LIN {X 0,Y 166.434,Z 455.503,A -85,B 0,C 180,E1 -24153.296,E2 -24153.296} C_VEL
LIN {X 0,Y 169.593,Z 462.541,A -85,B 0,C 180,E1 -24157.756,E2 -24157.756} C_VEL
LIN {X 0,Y 171.925,Z 468.212,A -85,B 0,C 180,E1 -24160.849,E2 -24160.849} C_VEL
LIN {X 0,Y 174.056,Z 474.701,A -85,B 0,C 180,E1 -24163.902,E2 -24163.902} C_VEL
LIN {X 0,Y 175.584,Z 481.015,A -85,B 0,C 180,E1 -24166.592,E2 -24166.592} C_VEL
LIN {X 0,Y 174.825,Z 487.861,A -85,B 0,C 180,E1 -24168.642,E2 -24168.642} C_VEL
LIN {X 0,Y 172.622,Z 497.216,A -85,B 0,C 180,E1 -24171.532,E2 -24171.532} C_VEL
LIN {X 0,Y 170.129,Z 504.353,A -85,B 0,C 180,E1 -24173.945,E2 -24173.945} C_VEL
LIN {X 0,Y 165.916,Z 511.785,A -85,B 0,C 180,E1 -24176.595,E2 -24176.595} C_VEL
LIN {X 0,Y 161.161,Z 519.066,A -85,B 0,C 180,E1 -24179.908,E2 -24179.908} C_VEL
LIN {X 0,Y 157.26,Z 524.869,A -85,B 0,C 180,E1 -24183.462,E2 -24183.462} C_VEL
LIN {X 0,Y 153.991,Z 529.408,A -85,B 0,C 180,E1 -24187.181,E2 -24187.181} C_VEL
LIN {X 0,Y 151.34,Z 532.851,A -85,B 0,C 180,E1 -24191.037,E2 -24191.037} C_VEL
LIN {X 0,Y 149.93,Z 534.573,A -85,B 0,C 180,E1 -24193.672,E2 -24193.672} C_VEL
LIN {X 0,Y 148.978,Z 535.901,A -85,B 0,C 180,E1 -24196.363,E2 -24196.363} C_VEL
LIN {X 0,Y 148.309,Z 536.803,A -85,B 0,C 180,E1 -24199.08,E2 -24199.08} C_VEL
LIN {X 0,Y 147.919,Z 537.372,A -85,B 0,C 180,E1 -24204.553,E2 -24204.553} C_VEL
LIN {X 0,Y 147.968,Z 537.384,A -85,B 0,C 180,E1 -24205.296,E2 -24205.296} C_VEL
LIN {X 0,Y 148.105,Z 541.561,A -85,B 0,C 180,E1 -24210.006,E2 -24210.006} C_VEL
LIN {X 0,Y 147.802,Z 543.506,A -85,B 0,C 180,E1 -24213.069,E2 -24213.069} C_VEL
LIN {X 0,Y 147.952,Z 545.577,A -85,B 0,C 180,E1 -24218.199,E2 -24218.199} C_VEL
LIN {X 0,Y 149.306,Z 546.349,A -85,B 0,C 180,E1 -24223.618,E2 -24223.618} C_VEL
LIN {X 0,Y 151.84,Z 545.71,A -85,B 0,C 180,E1 -24228.911,E2 -24228.911} C_VEL
LIN {X 0,Y 155.965,Z 543.606,A -85,B 0,C 180,E1 -24233.931,E2 -24233.931} C_VEL
LIN {X 0,Y 161.202,Z 540.049,A -85,B 0,C 180,E1 -24238.663,E2 -24238.663} C_VEL
LIN {X 0,Y 165.955,Z 536.223,A -85,B 0,C 180,E1 -24242.114,E2 -24242.114} C_VEL
LIN {X 0,Y 171.027,Z 531.735,A -85,B 0,C 180,E1 -24245.126,E2 -24245.126} C_VEL
LIN {X 0,Y 177.232,Z 525.759,A -85,B 0,C 180,E1 -24248.092,E2 -24248.092} C_VEL
LIN {X 0,Y 179.758,Z 522.779,A -85,B 0,C 180,E1 -24249.524,E2 -24249.524} C_VEL
LIN {X 0,Y 182.55,Z 517.989,A -85,B 0,C 180,E1 -24252.134,E2 -24252.134} C_VEL
LIN {X 0,Y 185.7,Z 511.799,A -85,B 0,C 180,E1 -24255.202,E2 -24255.202} C_VEL
LIN {X 0,Y 187.148,Z 509.452,A -85,B 0,C 180,E1 -24256.096,E2 -24256.096} C_VEL
LIN {X 0,Y 188.812,Z 506.875,A -85,B 0,C 180,E1 -24257.01,E2 -24257.01} C_VEL
LIN {X 0,Y 189.502,Z 504.868,A -85,B 0,C 180,E1 -24258.12,E2 -24258.12} C_VEL
LIN {X 0,Y 189.981,Z 501.234,A -85,B 0,C 180,E1 -24261.031,E2 -24261.031} C_VEL
LIN {X 0,Y 189.707,Z 499.154,A -85,B 0,C 180,E1 -24263.647,E2 -24263.647} C_VEL
LIN {X 0,Y 189.489,Z 497.804,A -85,B 0,C 180,E1 -24266.196,E2 -24266.196} C_VEL
LIN {X 0,Y 189.328,Z 496.956,A -85,B 0,C 180,E1 -24268.688,E2 -24268.688} C_VEL
LIN {X 0,Y 189.184,Z 496.682,A -85,B 0,C 180,E1 -24271.122,E2 -24271.122} C_VEL
LIN {X 0,Y 188.92,Z 497.163,A -85,B 0,C 180,E1 -24273.485,E2 -24273.485} C_VEL
LIN {X 0,Y 188.706,Z 498.014,A -85,B 0,C 180,E1 -24275.815,E2 -24275.815} C_VEL
LIN {X 0,Y 188.644,Z 499.613,A -85,B 0,C 180,E1 -24278.661,E2 -24278.661} C_VEL
LIN {X 0,Y 188.327,Z 502.026,A -85,B 0,C 180,E1 -24281.505,E2 -24281.505} C_VEL
LIN {X 0,Y 187.812,Z 504.455,A -85,B 0,C 180,E1 -24283.7,E2 -24283.7} C_VEL
LIN {X 0,Y 187.108,Z 506.134,A -85,B 0,C 180,E1 -24284.755,E2 -24284.755} C_VEL
LIN {X 0,Y 183.978,Z 511.853,A -85,B 0,C 180,E1 -24287.871,E2 -24287.871} C_VEL
LIN {X 0,Y 183.305,Z 512.868,A -85,B 0,C 180,E1 -24288.387,E2 -24288.387} C_VEL
LIN {X 0,Y 175.523,Z 520.816,A -85,B 0,C 180,E1 -24291.364,E2 -24291.364} C_VEL
LIN {X 0,Y 169.603,Z 526.103,A -85,B 0,C 180,E1 -24294.032,E2 -24294.032} C_VEL
LIN {X 0,Y 162.956,Z 531.203,A -85,B 0,C 180,E1 -24297.527,E2 -24297.527} C_VEL
LIN {X 0,Y 157.198,Z 535.016,A -85,B 0,C 180,E1 -24301.28,E2 -24301.28} C_VEL
LIN {X 0,Y 152.28,Z 537.685,A -85,B 0,C 180,E1 -24305.295,E2 -24305.295} C_VEL
LIN {X 0,Y 149.19,Z 538.988,A -85,B 0,C 180,E1 -24308.374,E2 -24308.374} C_VEL
LIN {X 0,Y 146.941,Z 539.635,A -85,B 0,C 180,E1 -24311.029,E2 -24311.029} C_VEL
LIN {X 0,Y 144.854,Z 539.91,A -85,B 0,C 180,E1 -24314.038,E2 -24314.038} C_VEL
LIN {X 0,Y 143.177,Z 539.754,A -85,B 0,C 180,E1 -24317.128,E2 -24317.128} C_VEL
LIN {X 0,Y 141.877,Z 539.109,A -85,B 0,C 180,E1 -24320.288,E2 -24320.288} C_VEL
LIN {X 0,Y 140.475,Z 536.929,A -85,B 0,C 180,E1 -24325.759,E2 -24325.759} C_VEL
LIN {X 0,Y 140.134,Z 533.138,A -85,B 0,C 180,E1 -24331.496,E2 -24331.496} C_VEL
LIN {X 0,Y 140.646,Z 527.91,A -85,B 0,C 180,E1 -24336.908,E2 -24336.908} C_VEL
LIN {X 0,Y 141.633,Z 521.475,A -85,B 0,C 180,E1 -24341.891,E2 -24341.891} C_VEL
LIN {X 0,Y 143.083,Z 513.619,A -85,B 0,C 180,E1 -24346.548,E2 -24346.548} C_VEL
LIN {X 0,Y 144.81,Z 505.438,A -85,B 0,C 180,E1 -24350.393,E2 -24350.393} C_VEL
LIN {X 0,Y 146.926,Z 496.371,A -85,B 0,C 180,E1 -24353.82,E2 -24353.82} C_VEL
LIN {X 0,Y 149.55,Z 484.775,A -85,B 0,C 180,E1 -24357.284,E2 -24357.284} C_VEL
LIN {X 0,Y 150.844,Z 478.491,A -85,B 0,C 180,E1 -24358.834,E2 -24358.834} C_VEL
LIN {X 0,Y 149.746,Z 466.485,A -85,B 0,C 180,E1 -24361.622,E2 -24361.622} C_VEL
LIN {X 0,Y 148.306,Z 454.178,A -85,B 0,C 180,E1 -24363.996,E2 -24363.996} C_VEL
LIN {X 0,Y 146.033,Z 439.457,A -85,B 0,C 180,E1 -24366.272,E2 -24366.272} C_VEL
LIN {X 0,Y 144.595,Z 431.334,A -85,B 0,C 180,E1 -24367.355,E2 -24367.355} C_VEL
LIN {X 0,Y 144.497,Z 428.599,A -85,B 0,C 180,E1 -24370.089,E2 -24370.089} C_VEL
LIN {X 0,Y 143.779,Z 424.334,A -85,B 0,C 180,E1 -24374.762,E2 -24374.762} C_VEL
LIN {X 0,Y 144.189,Z 426.576,A -85,B 0,C 180,E1 -24378.751,E2 -24378.751} C_VEL
LIN {X 0,Y 144.55,Z 428.254,A -85,B 0,C 180,E1 -24381.607,E2 -24381.607} C_VEL
LIN {X 0,Y 145.11,Z 431.41,A -85,B 0,C 180,E1 -24386.349,E2 -24386.349} C_VEL
LIN {X 0,Y 147.226,Z 438.421,A -85,B 0,C 180,E1 -24387.563,E2 -24387.563} C_VEL
LIN {X 0,Y 149.67,Z 450.103,A -85,B 0,C 180,E1 -24389.729,E2 -24389.729} C_VEL
LIN {X 0,Y 151.023,Z 459.538,A -85,B 0,C 180,E1 -24391.761,E2 -24391.761} C_VEL
LIN {X 0,Y 151.915,Z 469.677,A -85,B 0,C 180,E1 -24394.305,E2 -24394.305} C_VEL
LIN {X 0,Y 152.07,Z 476.634,A -85,B 0,C 180,E1 -24396.296,E2 -24396.296} C_VEL
LIN {X 0,Y 149.516,Z 486.319,A -85,B 0,C 180,E1 -24399.217,E2 -24399.217} C_VEL
LIN {X 0,Y 147.124,Z 494.539,A -85,B 0,C 180,E1 -24402.407,E2 -24402.407} C_VEL
LIN {X 0,Y 145.091,Z 501.591,A -85,B 0,C 180,E1 -24405.871,E2 -24405.871} C_VEL
LIN {X 0,Y 143.101,Z 508.264,A -85,B 0,C 180,E1 -24410.1,E2 -24410.1} C_VEL
LIN {X 0,Y 141.677,Z 513.845,A -85,B 0,C 180,E1 -24414.873,E2 -24414.873} C_VEL
LIN {X 0,Y 140.813,Z 517.925,A -85,B 0,C 180,E1 -24419.932,E2 -24419.932} C_VEL
LIN {X 0,Y 140.738,Z 519.778,A -85,B 0,C 180,E1 -24423.311,E2 -24423.311} C_VEL
LIN {X 0,Y 141.111,Z 521.102,A -85,B 0,C 180,E1 -24427.169,E2 -24427.169} C_VEL
LIN {X 0,Y 142.415,Z 521.578,A -85,B 0,C 180,E1 -24432.25,E2 -24432.25} C_VEL
LIN {X 0,Y 144.53,Z 520.651,A -85,B 0,C 180,E1 -24437.097,E2 -24437.097} C_VEL
LIN {X 0,Y 147.428,Z 518.388,A -85,B 0,C 180,E1 -24441.706,E2 -24441.706} C_VEL
LIN {X 0,Y 151.032,Z 514.814,A -85,B 0,C 180,E1 -24446.056,E2 -24446.056} C_VEL
LIN {X 0,Y 155.463,Z 509.711,A -85,B 0,C 180,E1 -24450.181,E2 -24450.181} C_VEL
LIN {X 0,Y 159.597,Z 504.413,A -85,B 0,C 180,E1 -24453.282,E2 -24453.282} C_VEL
LIN {X 0,Y 164.694,Z 496.927,A -85,B 0,C 180,E1 -24456.542,E2 -24456.542} C_VEL
LIN {X 0,Y 166.412,Z 493.936,A -85,B 0,C 180,E1 -24457.661,E2 -24457.661} C_VEL
LIN {X 0,Y 167.735,Z 487.888,A -85,B 0,C 180,E1 -24460.416,E2 -24460.416} C_VEL
LIN {X 0,Y 168.468,Z 480.689,A -85,B 0,C 180,E1 -24463.612,E2 -24463.612} C_VEL
LIN {X 0,Y 168.234,Z 475.376,A -85,B 0,C 180,E1 -24466.102,E2 -24466.102} C_VEL
LIN {X 0,Y 167.124,Z 469.966,A -85,B 0,C 180,E1 -24469.093,E2 -24469.093} C_VEL
LIN {X 0,Y 165.277,Z 464.338,A -85,B 0,C 180,E1 -24472.672,E2 -24472.672} C_VEL
LIN {X 0,Y 163.325,Z 459.565,A -85,B 0,C 180,E1 -24476.343,E2 -24476.343} C_VEL
LIN {X 0,Y 160.83,Z 453.807,A -85,B 0,C 180,E1 -24481.879,E2 -24481.879} C_VEL
LIN {X 0,Y 157.948,Z 450.631,A -85,B 0,C 180,E1 -24490.253,E2 -24490.253} C_VEL
LIN {X 0,Y 157.668,Z 450.184,A -85,B 0,C 180,E1 -24492.879,E2 -24492.879} C_VEL
LIN {X 0,Y 157.604,Z 450.264,A -85,B 0,C 180,E1 -24495.52,E2 -24495.52} C_VEL
LIN {X 0,Y 157.752,Z 450.92,A -85,B 0,C 180,E1 -24498.172,E2 -24498.172} C_VEL
LIN {X 0,Y 158.774,Z 453.562,A -85,B 0,C 180,E1 -24503.478,E2 -24503.478} C_VEL
LIN {X 0,Y 160.478,Z 455.834,A -85,B 0,C 180,E1 -24507.378,E2 -24507.378} C_VEL
LIN {X 0,Y 163.34,Z 462.175,A -85,B 0,C 180,E1 -24513.073,E2 -24513.073} C_VEL
LIN {X 0,Y 165.352,Z 467.137,A -85,B 0,C 180,E1 -24516.517,E2 -24516.517} C_VEL
LIN {X 0,Y 167.729,Z 474.013,A -85,B 0,C 180,E1 -24520.504,E2 -24520.504} C_VEL
LIN {X 0,Y 169.286,Z 479.911,A -85,B 0,C 180,E1 -24523.449,E2 -24523.449} C_VEL
LIN {X 0,Y 170.103,Z 484.114,A -85,B 0,C 180,E1 -24525.391,E2 -24525.391} C_VEL
LIN {X 0,Y 169.683,Z 487.961,A -85,B 0,C 180,E1 -24526.705,E2 -24526.705} C_VEL
LIN {X 0,Y 167.552,Z 496.578,A -85,B 0,C 180,E1 -24529.499,E2 -24529.499} C_VEL
LIN {X 0,Y 164.427,Z 505,A -85,B 0,C 180,E1 -24532.485,E2 -24532.485} C_VEL
LIN {X 0,Y 160.933,Z 510.894,A -85,B 0,C 180,E1 -24534.653,E2 -24534.653} C_VEL
LIN {X 0,Y 155.821,Z 518.232,A -85,B 0,C 180,E1 -24538.005,E2 -24538.005} C_VEL
LIN {X 0,Y 150.892,Z 524.956,A -85,B 0,C 180,E1 -24542.248,E2 -24542.248} C_VEL
LIN {X 0,Y 147.452,Z 529.377,A -85,B 0,C 180,E1 -24546.108,E2 -24546.108} C_VEL
LIN {X 0,Y 144.62,Z 532.715,A -85,B 0,C 180,E1 -24550.12,E2 -24550.12} C_VEL
LIN {X 0,Y 143.092,Z 534.383,A -85,B 0,C 180,E1 -24552.868,E2 -24552.868} C_VEL
LIN {X 0,Y 142.042,Z 535.645,A -85,B 0,C 180,E1 -24555.684,E2 -24555.684} C_VEL
LIN {X 0,Y 140.9,Z 536.888,A -85,B 0,C 180,E1 -24561.401,E2 -24561.401} C_VEL
LIN {X 0,Y 140.926,Z 537.009,A -85,B 0,C 180,E1 -24565.683,E2 -24565.683} C_VEL
LIN {X 0,Y 141.044,Z 540.777,A -85,B 0,C 180,E1 -24570.006,E2 -24570.006} C_VEL
LIN {X 0,Y 140.746,Z 544.03,A -85,B 0,C 180,E1 -24575.738,E2 -24575.738} C_VEL
LIN {X 0,Y 141.489,Z 545.788,A -85,B 0,C 180,E1 -24581.466,E2 -24581.466} C_VEL
LIN {X 0,Y 143.556,Z 546.056,A -85,B 0,C 180,E1 -24587.088,E2 -24587.088} C_VEL
LIN {X 0,Y 147.13,Z 544.937,A -85,B 0,C 180,E1 -24592.472,E2 -24592.472} C_VEL
LIN {X 0,Y 152.123,Z 542.393,A -85,B 0,C 180,E1 -24597.522,E2 -24597.522} C_VEL
LIN {X 0,Y 158.161,Z 538.375,A -85,B 0,C 180,E1 -24602.23,E2 -24602.23} C_VEL
LIN {X 0,Y 165.332,Z 532.771,A -85,B 0,C 180,E1 -24606.527,E2 -24606.527} C_VEL
LIN {X 0,Y 173.738,Z 525.291,A -85,B 0,C 180,E1 -24610.339,E2 -24610.339} C_VEL
LIN {X 0,Y 181.682,Z 517.009,A -85,B 0,C 180,E1 -24613.369,E2 -24613.369} C_VEL
LIN {X 0,Y 187.148,Z 509.452,A -85,B 0,C 180,E1 -24616.096,E2 -24616.096} C_VEL
LIN {X 0,Y 188.189,Z 507.429,A -85,B 0,C 180,E1 -24617.029,E2 -24617.029} C_VEL
LIN {X 0,Y 188.45,Z 505.993,A -85,B 0,C 180,E1 -24618.115,E2 -24618.115} C_VEL
LIN {X 0,Y 187.888,Z 504.71,A -85,B 0,C 180,E1 -24619.879,E2 -24619.879} C_VEL
LIN {X 0,Y 185.048,Z 503.736,A -85,B 0,C 180,E1 -24624.404,E2 -24624.404} C_VEL
LIN {X 0,Y 184.695,Z 503.307,A -85,B 0,C 180,E1 -24625.736,E2 -24625.736} C_VEL
LIN {X 0,Y 184.575,Z 502.51,A -85,B 0,C 180,E1 -24627.786,E2 -24627.786} C_VEL
LIN {X 0,Y 184.432,Z 501.995,A -85,B 0,C 180,E1 -24631.224,E2 -24631.224} C_VEL
LIN {X 0,Y 183.919,Z 502.999,A -85,B 0,C 180,E1 -24635.143,E2 -24635.143} C_VEL
LIN {X 0,Y 183.755,Z 504.095,A -85,B 0,C 180,E1 -24637.513,E2 -24637.513} C_VEL
LIN {X 0,Y 183.185,Z 506.581,A -85,B 0,C 180,E1 -24640.966,E2 -24640.966} C_VEL
LIN {X 0,Y 182.92,Z 507.664,A -85,B 0,C 180,E1 -24642.098,E2 -24642.098} C_VEL
LIN {X 0,Y 182.361,Z 508.953,A -85,B 0,C 180,E1 -24643.199,E2 -24643.199} C_VEL
LIN {X 0,Y 180.23,Z 512.392,A -85,B 0,C 180,E1 -24645.317,E2 -24645.317} C_VEL
LIN {X 0,Y 178.364,Z 515.141,A -85,B 0,C 180,E1 -24646.904,E2 -24646.904} C_VEL
LIN {X 0,Y 170.622,Z 522.314,A -85,B 0,C 180,E1 -24649.744,E2 -24649.744} C_VEL
LIN {X 0,Y 162.801,Z 528.59,A -85,B 0,C 180,E1 -24653.201,E2 -24653.201} C_VEL
LIN {X 0,Y 157.134,Z 532.454,A -85,B 0,C 180,E1 -24656.152,E2 -24656.152} C_VEL
LIN {X 0,Y 151.083,Z 535.98,A -85,B 0,C 180,E1 -24659.999,E2 -24659.999} C_VEL
LIN {X 0,Y 147.516,Z 537.697,A -85,B 0,C 180,E1 -24662.73,E2 -24662.73} C_VEL
LIN {X 0,Y 141.971,Z 539.667,A -85,B 0,C 180,E1 -24668.049,E2 -24668.049} C_VEL
LIN {X 0,Y 137.613,Z 540.109,A -85,B 0,C 180,E1 -24673.968,E2 -24673.968} C_VEL
LIN {X 0,Y 134.76,Z 538.93,A -85,B 0,C 180,E1 -24680.144,E2 -24680.144} C_VEL
LIN {X 0,Y 133.305,Z 536.181,A -85,B 0,C 180,E1 -24686.317,E2 -24686.317} C_VEL
LIN {X 0,Y 133.078,Z 531.96,A -85,B 0,C 180,E1 -24692.32,E2 -24692.32} C_VEL
LIN {X 0,Y 133.53,Z 527.733,A -85,B 0,C 180,E1 -24696.685,E2 -24696.685} C_VEL
LIN {X 0,Y 134.514,Z 521.399,A -85,B 0,C 180,E1 -24701.77,E2 -24701.77} C_VEL
LIN {X 0,Y 135.85,Z 513.969,A -85,B 0,C 180,E1 -24706.407,E2 -24706.407} C_VEL
LIN {X 0,Y 137.667,Z 505.685,A -85,B 0,C 180,E1 -24710.536,E2 -24710.536} C_VEL
LIN {X 0,Y 139.814,Z 496.657,A -85,B 0,C 180,E1 -24714.148,E2 -24714.148} C_VEL
LIN {X 0,Y 142.439,Z 485.41,A -85,B 0,C 180,E1 -24717.704,E2 -24717.704} C_VEL
LIN {X 0,Y 143.815,Z 478.396,A -85,B 0,C 180,E1 -24719.529,E2 -24719.529} C_VEL
LIN {X 0,Y 142.755,Z 466.616,A -85,B 0,C 180,E1 -24722.393,E2 -24722.393} C_VEL
LIN {X 0,Y 141.42,Z 454.741,A -85,B 0,C 180,E1 -24724.79,E2 -24724.79} C_VEL
LIN {X 0,Y 139.283,Z 440.562,A -85,B 0,C 180,E1 -24727.099,E2 -24727.099} C_VEL
LIN {X 0,Y 137.609,Z 431.53,A -85,B 0,C 180,E1 -24728.365,E2 -24728.365} C_VEL
LIN {X 0,Y 137.213,Z 428.007,A -85,B 0,C 180,E1 -24732.096,E2 -24732.096} C_VEL
LIN {X 0,Y 136.825,Z 425.791,A -85,B 0,C 180,E1 -24734.636,E2 -24734.636} C_VEL
LIN {X 0,Y 137.532,Z 429.376,A -85,B 0,C 180,E1 -24741.175,E2 -24741.175} C_VEL
LIN {X 0,Y 137.868,Z 431.391,A -85,B 0,C 180,E1 -24744.601,E2 -24744.601} C_VEL
LIN {X 0,Y 139.322,Z 434.977,A -85,B 0,C 180,E1 -24745.367,E2 -24745.367} C_VEL
LIN {X 0,Y 141.065,Z 440.756,A -85,B 0,C 180,E1 -24746.493,E2 -24746.493} C_VEL
LIN {X 0,Y 143.374,Z 452.691,A -85,B 0,C 180,E1 -24748.939,E2 -24748.939} C_VEL
LIN {X 0,Y 144.738,Z 463.608,A -85,B 0,C 180,E1 -24751.536,E2 -24751.536} C_VEL
LIN {X 0,Y 145.317,Z 474.217,A -85,B 0,C 180,E1 -24754.501,E2 -24754.501} C_VEL
LIN {X 0,Y 145.23,Z 477.614,A -85,B 0,C 180,E1 -24755.548,E2 -24755.548} C_VEL
LIN {X 0,Y 142.664,Z 486.874,A -85,B 0,C 180,E1 -24758.492,E2 -24758.492} C_VEL
LIN {X 0,Y 139.841,Z 496.127,A -85,B 0,C 180,E1 -24762.326,E2 -24762.326} C_VEL
LIN {X 0,Y 137.573,Z 503.587,A -85,B 0,C 180,E1 -24766.37,E2 -24766.37} C_VEL
LIN {X 0,Y 135.584,Z 510.216,A -85,B 0,C 180,E1 -24771.091,E2 -24771.091} C_VEL
LIN {X 0,Y 134.33,Z 515.09,A -85,B 0,C 180,E1 -24775.843,E2 -24775.843} C_VEL
LIN {X 0,Y 133.733,Z 518.16,A -85,B 0,C 180,E1 -24779.942,E2 -24779.942} C_VEL
LIN {X 0,Y 133.765,Z 520.802,A -85,B 0,C 180,E1 -24785.297,E2 -24785.297} C_VEL
LIN {X 0,Y 134.319,Z 521.728,A -85,B 0,C 180,E1 -24788.884,E2 -24788.884} C_VEL
LIN {X 0,Y 135.717,Z 521.998,A -85,B 0,C 180,E1 -24793.534,E2 -24793.534} C_VEL
LIN {X 0,Y 138.117,Z 520.976,A -85,B 0,C 180,E1 -24798.587,E2 -24798.587} C_VEL
LIN {X 0,Y 141.308,Z 518.673,A -85,B 0,C 180,E1 -24803.359,E2 -24803.359} C_VEL
LIN {X 0,Y 145.265,Z 515.006,A -85,B 0,C 180,E1 -24807.848,E2 -24807.848} C_VEL
LIN {X 0,Y 150.096,Z 509.817,A -85,B 0,C 180,E1 -24812.081,E2 -24812.081} C_VEL
LIN {X 0,Y 154.673,Z 504.25,A -85,B 0,C 180,E1 -24815.317,E2 -24815.317} C_VEL
LIN {X 0,Y 160.53,Z 495.958,A -85,B 0,C 180,E1 -24818.888,E2 -24818.888} C_VEL
LIN {X 0,Y 162.059,Z 490.288,A -85,B 0,C 180,E1 -24821.677,E2 -24821.677} C_VEL
LIN {X 0,Y 163.059,Z 483.358,A -85,B 0,C 180,E1 -24825.014,E2 -24825.014} C_VEL
LIN {X 0,Y 163.037,Z 478.55,A -85,B 0,C 180,E1 -24827.554,E2 -24827.554} C_VEL
LIN {X 0,Y 161.843,Z 472.685,A -85,B 0,C 180,E1 -24831.259,E2 -24831.259} C_VEL
LIN {X 0,Y 160.949,Z 469.202,A -85,B 0,C 180,E1 -24833.734,E2 -24833.734} C_VEL
LIN {X 0,Y 159.399,Z 464.755,A -85,B 0,C 180,E1 -24837.474,E2 -24837.474} C_VEL
LIN {X 0,Y 157.642,Z 459.938,A -85,B 0,C 180,E1 -24842.556,E2 -24842.556} C_VEL
LIN {X 0,Y 155.384,Z 457.237,A -85,B 0,C 180,E1 -24850.424,E2 -24850.424} C_VEL
LIN {X 0,Y 155.171,Z 456.816,A -85,B 0,C 180,E1 -24853.09,E2 -24853.09} C_VEL
LIN {X 0,Y 155.13,Z 457.006,A -85,B 0,C 180,E1 -24855.774,E2 -24855.774} C_VEL
LIN {X 0,Y 155.254,Z 457.742,A -85,B 0,C 180,E1 -24858.475,E2 -24858.475} C_VEL
LIN {X 0,Y 157.398,Z 462.06,A -85,B 0,C 180,E1 -24866.76,E2 -24866.76} C_VEL
LIN {X 0,Y 159.766,Z 468.365,A -85,B 0,C 180,E1 -24872.696,E2 -24872.696} C_VEL
LIN {X 0,Y 161.646,Z 474.19,A -85,B 0,C 180,E1 -24876.832,E2 -24876.832} C_VEL
LIN {X 0,Y 163.267,Z 479.692,A -85,B 0,C 180,E1 -24880.219,E2 -24880.219} C_VEL
LIN {X 0,Y 164.418,Z 485.714,A -85,B 0,C 180,E1 -24883.402,E2 -24883.402} C_VEL
LIN {X 0,Y 164.603,Z 488.774,A -85,B 0,C 180,E1 -24884.829,E2 -24884.829} C_VEL
LIN {X 0,Y 162.395,Z 496.794,A -85,B 0,C 180,E1 -24887.609,E2 -24887.609} C_VEL
LIN {X 0,Y 159.563,Z 504.092,A -85,B 0,C 180,E1 -24890.317,E2 -24890.317} C_VEL
LIN {X 0,Y 157.151,Z 508.602,A -85,B 0,C 180,E1 -24892.062,E2 -24892.062} C_VEL
LIN {X 0,Y 151.57,Z 516.352,A -85,B 0,C 180,E1 -24895.397,E2 -24895.397} C_VEL
LIN {X 0,Y 147.483,Z 521.585,A -85,B 0,C 180,E1 -24898.395,E2 -24898.395} C_VEL
LIN {X 0,Y 143.713,Z 526.242,A -85,B 0,C 180,E1 -24901.897,E2 -24901.897} C_VEL
LIN {X 0,Y 139.861,Z 530.55,A -85,B 0,C 180,E1 -24906.304,E2 -24906.304} C_VEL
LIN {X 0,Y 137.945,Z 532.58,A -85,B 0,C 180,E1 -24909.114,E2 -24909.114} C_VEL
LIN {X 0,Y 136.292,Z 534.197,A -85,B 0,C 180,E1 -24911.985,E2 -24911.985} C_VEL
LIN {X 0,Y 134.322,Z 536.12,A -85,B 0,C 180,E1 -24917.927,E2 -24917.927} C_VEL
LIN {X 0,Y 133.854,Z 536.499,A -85,B 0,C 180,E1 -24920.944,E2 -24920.944} C_VEL
LIN {X 0,Y 133.889,Z 536.308,A -85,B 0,C 180,E1 -24925.832,E2 -24925.832} C_VEL
LIN {X 0,Y 133.983,Z 539.877,A -85,B 0,C 180,E1 -24930.007,E2 -24930.007} C_VEL
LIN {X 0,Y 133.72,Z 541.858,A -85,B 0,C 180,E1 -24933.019,E2 -24933.019} C_VEL
LIN {X 0,Y 133.943,Z 544.554,A -85,B 0,C 180,E1 -24939.063,E2 -24939.063} C_VEL
LIN {X 0,Y 135.483,Z 545.791,A -85,B 0,C 180,E1 -24945.039,E2 -24945.039} C_VEL
LIN {X 0,Y 138.468,Z 545.628,A -85,B 0,C 180,E1 -24950.818,E2 -24950.818} C_VEL
LIN {X 0,Y 143.089,Z 544.04,A -85,B 0,C 180,E1 -24956.241,E2 -24956.241} C_VEL
LIN {X 0,Y 148.929,Z 541.073,A -85,B 0,C 180,E1 -24961.278,E2 -24961.278} C_VEL
LIN {X 0,Y 153.776,Z 537.996,A -85,B 0,C 180,E1 -24964.648,E2 -24964.648} C_VEL
LIN {X 0,Y 159.739,Z 533.768,A -85,B 0,C 180,E1 -24968.027,E2 -24968.027} C_VEL
LIN {X 0,Y 166.248,Z 528.644,A -85,B 0,C 180,E1 -24970.945,E2 -24970.945} C_VEL
LIN {X 0,Y 174.4,Z 521.267,A -85,B 0,C 180,E1 -24974.044,E2 -24974.044} C_VEL
LIN {X 0,Y 177.84,Z 517.687,A -85,B 0,C 180,E1 -24975.349,E2 -24975.349} C_VEL
LIN {X 0,Y 183.011,Z 511.124,A -85,B 0,C 180,E1 -24977.838,E2 -24977.838} C_VEL
LIN {X 0,Y 184.001,Z 509.611,A -85,B 0,C 180,E1 -24978.482,E2 -24978.482} C_VEL
LIN {X 0,Y 184.504,Z 507.996,A -85,B 0,C 180,E1 -24979.642,E2 -24979.642} C_VEL
LIN {X 0,Y 184.815,Z 506.578,A -85,B 0,C 180,E1 -24980.933,E2 -24980.933} C_VEL
LIN {X 0,Y 184.926,Z 504.798,A -85,B 0,C 180,E1 -24982.955,E2 -24982.955} C_VEL
LIN {X 0,Y 184.695,Z 503.307,A -85,B 0,C 180,E1 -24985.736,E2 -24985.736} C_VEL
LIN {X 0,Y 184.093,Z 503.142,A -85,B 0,C 180,E1 -24987.559,E2 -24987.559} C_VEL
LIN {X 0,Y 182.876,Z 503.911,A -85,B 0,C 180,E1 -24989.363,E2 -24989.363} C_VEL
LIN {X 0,Y 179.151,Z 507.539,A -85,B 0,C 180,E1 -24994.22,E2 -24994.22} C_VEL
LIN {X 0,Y 178.754,Z 508.182,A -85,B 0,C 180,E1 -24995.496,E2 -24995.496} C_VEL
LIN {X 0,Y 178.617,Z 508.687,A -85,B 0,C 180,E1 -24996.829,E2 -24996.829} C_VEL
LIN {X 0,Y 178.191,Z 510.04,A -85,B 0,C 180,E1 -24999.208,E2 -24999.208} C_VEL
LIN {X 0,Y 177.492,Z 511.907,A -85,B 0,C 180,E1 -25001.531,E2 -25001.531} C_VEL
LIN {X 0,Y 176.68,Z 513.237,A -85,B 0,C 180,E1 -25002.641,E2 -25002.641} C_VEL
LIN {X 0,Y 173.493,Z 517.348,A -85,B 0,C 180,E1 -25005.333,E2 -25005.333} C_VEL
LIN {X 0,Y 165.05,Z 524.498,A -85,B 0,C 180,E1 -25008.36,E2 -25008.36} C_VEL
LIN {X 0,Y 156.048,Z 530.857,A -85,B 0,C 180,E1 -25012.264,E2 -25012.264} C_VEL
LIN {X 0,Y 151.393,Z 533.632,A -85,B 0,C 180,E1 -25014.672,E2 -25014.672} C_VEL
LIN {X 0,Y 147.114,Z 535.919,A -85,B 0,C 180,E1 -25017.261,E2 -25017.261} C_VEL
LIN {X 0,Y 140.654,Z 538.692,A -85,B 0,C 180,E1 -25021.955,E2 -25021.955} C_VEL
LIN {X 0,Y 134.757,Z 540.203,A -85,B 0,C 180,E1 -25027.692,E2 -25027.692} C_VEL
LIN {X 0,Y 130.339,Z 540.171,A -85,B 0,C 180,E1 -25033.91,E2 -25033.91} C_VEL
LIN {X 0,Y 127.509,Z 538.489,A -85,B 0,C 180,E1 -25040.43,E2 -25040.43} C_VEL
LIN {X 0,Y 126.131,Z 535.301,A -85,B 0,C 180,E1 -25046.923,E2 -25046.923} C_VEL
LIN {X 0,Y 125.977,Z 531.907,A -85,B 0,C 180,E1 -25051.691,E2 -25051.691} C_VEL
LIN {X 0,Y 126.578,Z 526.199,A -85,B 0,C 180,E1 -25057.643,E2 -25057.643} C_VEL
LIN {X 0,Y 127.718,Z 519.453,A -85,B 0,C 180,E1 -25062.975,E2 -25062.975} C_VEL
LIN {X 0,Y 129.053,Z 512.468,A -85,B 0,C 180,E1 -25067.321,E2 -25067.321} C_VEL
LIN {X 0,Y 131.034,Z 503.675,A -85,B 0,C 180,E1 -25071.688,E2 -25071.688} C_VEL
LIN {X 0,Y 133.377,Z 494.169,A -85,B 0,C 180,E1 -25075.462,E2 -25075.462} C_VEL
LIN {X 0,Y 136.004,Z 483.3,A -85,B 0,C 180,E1 -25078.879,E2 -25078.879} C_VEL
LIN {X 0,Y 136.784,Z 478.378,A -85,B 0,C 180,E1 -25080.206,E2 -25080.206} C_VEL
LIN {X 0,Y 135.756,Z 466.195,A -85,B 0,C 180,E1 -25083.302,E2 -25083.302} C_VEL
LIN {X 0,Y 134.388,Z 453.971,A -85,B 0,C 180,E1 -25085.874,E2 -25085.874} C_VEL
LIN {X 0,Y 132.271,Z 440.078,A -85,B 0,C 180,E1 -25088.261,E2 -25088.261} C_VEL
LIN {X 0,Y 130.572,Z 431.669,A -85,B 0,C 180,E1 -25089.514,E2 -25089.514} C_VEL
LIN {X 0,Y 129.898,Z 427.259,A -85,B 0,C 180,E1 -25094.48,E2 -25094.48} C_VEL
LIN {X 0,Y 130.516,Z 430.506,A -85,B 0,C 180,E1 -25100.697,E2 -25100.697} C_VEL
LIN {X 0,Y 130.674,Z 431.638,A -85,B 0,C 180,E1 -25102.752,E2 -25102.752} C_VEL
LIN {X 0,Y 132.142,Z 435.222,A -85,B 0,C 180,E1 -25103.595,E2 -25103.595} C_VEL
LIN {X 0,Y 134.561,Z 441.41,A -85,B 0,C 180,E1 -25105.032,E2 -25105.032} C_VEL
LIN {X 0,Y 136.861,Z 453.788,A -85,B 0,C 180,E1 -25107.73,E2 -25107.73} C_VEL
LIN {X 0,Y 137.937,Z 462.783,A -85,B 0,C 180,E1 -25109.994,E2 -25109.994} C_VEL
LIN {X 0,Y 138.556,Z 472.831,A -85,B 0,C 180,E1 -25112.901,E2 -25112.901} C_VEL
LIN {X 0,Y 138.425,Z 478.513,A -85,B 0,C 180,E1 -25114.726,E2 -25114.726} C_VEL
LIN {X 0,Y 135.54,Z 488.224,A -85,B 0,C 180,E1 -25118.023,E2 -25118.023} C_VEL
LIN {X 0,Y 133.075,Z 496.005,A -85,B 0,C 180,E1 -25121.416,E2 -25121.416} C_VEL
LIN {X 0,Y 130.713,Z 503.484,A -85,B 0,C 180,E1 -25125.587,E2 -25125.587} C_VEL
LIN {X 0,Y 128.729,Z 509.804,A -85,B 0,C 180,E1 -25130.214,E2 -25130.214} C_VEL
LIN {X 0,Y 127.526,Z 514.191,A -85,B 0,C 180,E1 -25134.406,E2 -25134.406} C_VEL
LIN {X 0,Y 126.648,Z 518.393,A -85,B 0,C 180,E1 -25139.953,E2 -25139.953} C_VEL
LIN {X 0,Y 126.554,Z 520.376,A -85,B 0,C 180,E1 -25143.724,E2 -25143.724} C_VEL
LIN {X 0,Y 127.319,Z 522.086,A -85,B 0,C 180,E1 -25149.396,E2 -25149.396} C_VEL
LIN {X 0,Y 129.123,Z 522.396,A -85,B 0,C 180,E1 -25155.027,E2 -25155.027} C_VEL
LIN {X 0,Y 131.812,Z 521.31,A -85,B 0,C 180,E1 -25160.223,E2 -25160.223} C_VEL
LIN {X 0,Y 135.887,Z 518.496,A -85,B 0,C 180,E1 -25165.83,E2 -25165.83} C_VEL
LIN {X 0,Y 139.682,Z 515.195,A -85,B 0,C 180,E1 -25169.793,E2 -25169.793} C_VEL
LIN {X 0,Y 144.967,Z 509.92,A -85,B 0,C 180,E1 -25174.132,E2 -25174.132} C_VEL
LIN {X 0,Y 149.983,Z 504.121,A -85,B 0,C 180,E1 -25177.49,E2 -25177.49} C_VEL
LIN {X 0,Y 154.677,Z 497.943,A -85,B 0,C 180,E1 -25180.209,E2 -25180.209} C_VEL
LIN {X 0,Y 156.141,Z 493.743,A -85,B 0,C 180,E1 -25182.436,E2 -25182.436} C_VEL
LIN {X 0,Y 157.574,Z 487.345,A -85,B 0,C 180,E1 -25185.801,E2 -25185.801} C_VEL
LIN {X 0,Y 157.888,Z 482.991,A -85,B 0,C 180,E1 -25188.281,E2 -25188.281} C_VEL
LIN {X 0,Y 157.117,Z 477.195,A -85,B 0,C 180,E1 -25192.289,E2 -25192.289} C_VEL
LIN {X 0,Y 156.027,Z 472.537,A -85,B 0,C 180,E1 -25196.127,E2 -25196.127} C_VEL
LIN {X 0,Y 154.895,Z 468.749,A -85,B 0,C 180,E1 -25200.001,E2 -25200.001} C_VEL
LIN {X 0,Y 154.3,Z 466.442,A -85,B 0,C 180,E1 -25202.611,E2 -25202.611} C_VEL
LIN {X 0,Y 152.464,Z 463.674,A -85,B 0,C 180,E1 -25210.626,E2 -25210.626} C_VEL
LIN {X 0,Y 152.243,Z 463.371,A -85,B 0,C 180,E1 -25214.235,E2 -25214.235} C_VEL
LIN {X 0,Y 152.269,Z 463.598,A -85,B 0,C 180,E1 -25216.078,E2 -25216.078} C_VEL
LIN {X 0,Y 152.364,Z 464.452,A -85,B 0,C 180,E1 -25218.838,E2 -25218.838} C_VEL
LIN {X 0,Y 153.324,Z 467.173,A -85,B 0,C 180,E1 -25224.365,E2 -25224.365} C_VEL
LIN {X 0,Y 154.196,Z 468.985,A -85,B 0,C 180,E1 -25227.116,E2 -25227.116} C_VEL
LIN {X 0,Y 155.54,Z 473.07,A -85,B 0,C 180,E1 -25231.306,E2 -25231.306} C_VEL
LIN {X 0,Y 157.302,Z 479.828,A -85,B 0,C 180,E1 -25236.478,E2 -25236.478} C_VEL
LIN {X 0,Y 158.571,Z 485.64,A -85,B 0,C 180,E1 -25240.221,E2 -25240.221} C_VEL
LIN {X 0,Y 159.132,Z 491.021,A -85,B 0,C 180,E1 -25243.252,E2 -25243.252} C_VEL
LIN {X 0,Y 158.588,Z 493.607,A -85,B 0,C 180,E1 -25244.297,E2 -25244.297} C_VEL
LIN {X 0,Y 155.575,Z 501.704,A -85,B 0,C 180,E1 -25247.351,E2 -25247.351} C_VEL
LIN {X 0,Y 152.552,Z 507.763,A -85,B 0,C 180,E1 -25249.845,E2 -25249.845} C_VEL
LIN {X 0,Y 146.731,Z 515.568,A -85,B 0,C 180,E1 -25253.231,E2 -25253.231} C_VEL
LIN {X 0,Y 141.493,Z 521.784,A -85,B 0,C 180,E1 -25256.89,E2 -25256.89} C_VEL
LIN {X 0,Y 137.168,Z 526.639,A -85,B 0,C 180,E1 -25260.803,E2 -25260.803} C_VEL
LIN {X 0,Y 133.363,Z 530.5,A -85,B 0,C 180,E1 -25265.073,E2 -25265.073} C_VEL
LIN {X 0,Y 131.32,Z 532.467,A -85,B 0,C 180,E1 -25268.007,E2 -25268.007} C_VEL
LIN {X 0,Y 129.535,Z 533.982,A -85,B 0,C 180,E1 -25271.01,E2 -25271.01} C_VEL
LIN {X 0,Y 127.354,Z 535.782,A -85,B 0,C 180,E1 -25277.255,E2 -25277.255} C_VEL
LIN {X 0,Y 126.83,Z 536.09,A -85,B 0,C 180,E1 -25280.438,E2 -25280.438} C_VEL
LIN {X 0,Y 126.842,Z 535.653,A -85,B 0,C 180,E1 -25286.116,E2 -25286.116} C_VEL
LIN {X 0,Y 126.924,Z 538.941,A -85,B 0,C 180,E1 -25290.007,E2 -25290.007} C_VEL
LIN {X 0,Y 126.68,Z 541.03,A -85,B 0,C 180,E1 -25293.187,E2 -25293.187} C_VEL
LIN {X 0,Y 126.937,Z 543.981,A -85,B 0,C 180,E1 -25299.568,E2 -25299.568} C_VEL
LIN {X 0,Y 128.619,Z 545.434,A -85,B 0,C 180,E1 -25305.862,E2 -25305.862} C_VEL
LIN {X 0,Y 131.855,Z 545.514,A -85,B 0,C 180,E1 -25311.914,E2 -25311.914} C_VEL
LIN {X 0,Y 136.744,Z 544.234,A -85,B 0,C 180,E1 -25317.559,E2 -25317.559} C_VEL
LIN {X 0,Y 142.926,Z 541.513,A -85,B 0,C 180,E1 -25322.751,E2 -25322.751} C_VEL
LIN {X 0,Y 150.227,Z 537.396,A -85,B 0,C 180,E1 -25327.464,E2 -25327.464} C_VEL
LIN {X 0,Y 156.485,Z 533.231,A -85,B 0,C 180,E1 -25330.64,E2 -25330.64} C_VEL
LIN {X 0,Y 163.372,Z 528.096,A -85,B 0,C 180,E1 -25333.501,E2 -25333.501} C_VEL
LIN {X 0,Y 171.956,Z 520.721,A -85,B 0,C 180,E1 -25336.513,E2 -25336.513} C_VEL
LIN {X 0,Y 178.389,Z 513.593,A -85,B 0,C 180,E1 -25339.363,E2 -25339.363} C_VEL
LIN {X 0,Y 179.01,Z 512.522,A -85,B 0,C 180,E1 -25340.034,E2 -25340.034} C_VEL
LIN {X 0,Y 179.52,Z 510.932,A -85,B 0,C 180,E1 -25341.54,E2 -25341.54} C_VEL
LIN {X 0,Y 179.677,Z 509.137,A -85,B 0,C 180,E1 -25344.075,E2 -25344.075} C_VEL
LIN {X 0,Y 179.594,Z 507.887,A -85,B 0,C 180,E1 -25346.779,E2 -25346.779} C_VEL
LIN {X 0,Y 179.476,Z 507.248,A -85,B 0,C 180,E1 -25349.491,E2 -25349.491} C_VEL
LIN {X 0,Y 179.29,Z 507.163,A -85,B 0,C 180,E1 -25351.94,E2 -25351.94} C_VEL
LIN {X 0,Y 178.754,Z 508.182,A -85,B 0,C 180,E1 -25355.496,E2 -25355.496} C_VEL
LIN {X 0,Y 178.11,Z 509.124,A -85,B 0,C 180,E1 -25356.704,E2 -25356.704} C_VEL
LIN {X 0,Y 176.799,Z 510.684,A -85,B 0,C 180,E1 -25357.811,E2 -25357.811} C_VEL
LIN {X 0,Y 172.261,Z 515.527,A -85,B 0,C 180,E1 -25360.65,E2 -25360.65} C_VEL
LIN {X 0,Y 171.363,Z 516.563,A -85,B 0,C 180,E1 -25361.435,E2 -25361.435} C_VEL
LIN {X 0,Y 169.464,Z 518.803,A -85,B 0,C 180,E1 -25363.123,E2 -25363.123} C_VEL
LIN {X 0,Y 168.323,Z 519.924,A -85,B 0,C 180,E1 -25363.82,E2 -25363.82} C_VEL
LIN {X 0,Y 161.461,Z 525.208,A -85,B 0,C 180,E1 -25366.148,E2 -25366.148} C_VEL
LIN {X 0,Y 153.267,Z 530.661,A -85,B 0,C 180,E1 -25369.43,E2 -25369.43} C_VEL
LIN {X 0,Y 145.759,Z 534.813,A -85,B 0,C 180,E1 -25373.076,E2 -25373.076} C_VEL
LIN {X 0,Y 139.135,Z 537.753,A -85,B 0,C 180,E1 -25377.104,E2 -25377.104} C_VEL
LIN {X 0,Y 133.578,Z 539.59,A -85,B 0,C 180,E1 -25381.283,E2 -25381.283} C_VEL
LIN {X 0,Y 127.549,Z 540.6,A -85,B 0,C 180,E1 -25387.297,E2 -25387.297} C_VEL
LIN {X 0,Y 123.069,Z 540.047,A -85,B 0,C 180,E1 -25393.854,E2 -25393.854} C_VEL
LIN {X 0,Y 120.309,Z 537.989,A -85,B 0,C 180,E1 -25400.517,E2 -25400.517} C_VEL
LIN {X 0,Y 118.991,Z 534.238,A -85,B 0,C 180,E1 -25407.618,E2 -25407.618} C_VEL
LIN {X 0,Y 118.922,Z 530.884,A -85,B 0,C 180,E1 -25412.131,E2 -25412.131} C_VEL
LIN {X 0,Y 119.57,Z 525.176,A -85,B 0,C 180,E1 -25418.108,E2 -25418.108} C_VEL
LIN {X 0,Y 120.667,Z 518.886,A -85,B 0,C 180,E1 -25423.182,E2 -25423.182} C_VEL
LIN {X 0,Y 122.284,Z 510.771,A -85,B 0,C 180,E1 -25428.342,E2 -25428.342} C_VEL
LIN {X 0,Y 124.438,Z 501.704,A -85,B 0,C 180,E1 -25432.914,E2 -25432.914} C_VEL
LIN {X 0,Y 126.958,Z 491.714,A -85,B 0,C 180,E1 -25436.851,E2 -25436.851} C_VEL
LIN {X 0,Y 129.805,Z 479.904,A -85,B 0,C 180,E1 -25440.505,E2 -25440.505} C_VEL
LIN {X 0,Y 128.957,Z 468.205,A -85,B 0,C 180,E1 -25443.71,E2 -25443.71} C_VEL
LIN {X 0,Y 127.756,Z 456.1,A -85,B 0,C 180,E1 -25446.488,E2 -25446.488} C_VEL
LIN {X 0,Y 125.9,Z 443.054,A -85,B 0,C 180,E1 -25448.932,E2 -25448.932} C_VEL
LIN {X 0,Y 124.303,Z 434.7,A -85,B 0,C 180,E1 -25450.27,E2 -25450.27} C_VEL
LIN {X 0,Y 123.429,Z 431.824,A -85,B 0,C 180,E1 -25450.774,E2 -25450.774} C_VEL
LIN {X 0,Y 122.982,Z 428.791,A -85,B 0,C 180,E1 -25454.449,E2 -25454.449} C_VEL
LIN {X 0,Y 123.581,Z 432.011,A -85,B 0,C 180,E1 -25460.738,E2 -25460.738} C_VEL
LIN {X 0,Y 124.959,Z 435.43,A -85,B 0,C 180,E1 -25461.584,E2 -25461.584} C_VEL
LIN {X 0,Y 128.493,Z 443.884,A -85,B 0,C 180,E1 -25463.85,E2 -25463.85} C_VEL
LIN {X 0,Y 130.448,Z 455.463,A -85,B 0,C 180,E1 -25466.59,E2 -25466.59} C_VEL
LIN {X 0,Y 131.418,Z 464.305,A -85,B 0,C 180,E1 -25468.985,E2 -25468.985} C_VEL
LIN {X 0,Y 131.899,Z 473.75,A -85,B 0,C 180,E1 -25471.902,E2 -25471.902} C_VEL
LIN {X 0,Y 131.658,Z 479.408,A -85,B 0,C 180,E1 -25473.819,E2 -25473.819} C_VEL
LIN {X 0,Y 128.958,Z 488.078,A -85,B 0,C 180,E1 -25476.893,E2 -25476.893} C_VEL
LIN {X 0,Y 126.368,Z 495.86,A -85,B 0,C 180,E1 -25480.406,E2 -25480.406} C_VEL
LIN {X 0,Y 124.253,Z 502.229,A -85,B 0,C 180,E1 -25484.017,E2 -25484.017} C_VEL
LIN {X 0,Y 122.166,Z 508.413,A -85,B 0,C 180,E1 -25488.437,E2 -25488.437} C_VEL
LIN {X 0,Y 120.46,Z 514.296,A -85,B 0,C 180,E1 -25494.096,E2 -25494.096} C_VEL
LIN {X 0,Y 119.539,Z 518.618,A -85,B 0,C 180,E1 -25499.996,E2 -25499.996} C_VEL
LIN {X 0,Y 119.621,Z 521.396,A -85,B 0,C 180,E1 -25505.971,E2 -25505.971} C_VEL
LIN {X 0,Y 120.488,Z 522.574,A -85,B 0,C 180,E1 -25510.689,E2 -25510.689} C_VEL
LIN {X 0,Y 122.569,Z 522.796,A -85,B 0,C 180,E1 -25516.524,E2 -25516.524} C_VEL
LIN {X 0,Y 125.609,Z 521.653,A -85,B 0,C 180,E1 -25522.016,E2 -25522.016} C_VEL
LIN {X 0,Y 129.49,Z 519.246,A -85,B 0,C 180,E1 -25527.13,E2 -25527.13} C_VEL
LIN {X 0,Y 134.315,Z 515.405,A -85,B 0,C 180,E1 -25531.907,E2 -25531.907} C_VEL
LIN {X 0,Y 140.04,Z 510.027,A -85,B 0,C 180,E1 -25536.33,E2 -25536.33} C_VEL
LIN {X 0,Y 145.012,Z 504.617,A -85,B 0,C 180,E1 -25539.482,E2 -25539.482} C_VEL
LIN {X 0,Y 149.309,Z 499.198,A -85,B 0,C 180,E1 -25542.001,E2 -25542.001} C_VEL
LIN {X 0,Y 151.314,Z 493.691,A -85,B 0,C 180,E1 -25545.202,E2 -25545.202} C_VEL
LIN {X 0,Y 152.395,Z 489.119,A -85,B 0,C 180,E1 -25547.852,E2 -25547.852} C_VEL
LIN {X 0,Y 152.601,Z 486.768,A -85,B 0,C 180,E1 -25549.385,E2 -25549.385} C_VEL
LIN {X 0,Y 152.256,Z 481.584,A -85,B 0,C 180,E1 -25553.374,E2 -25553.374} C_VEL
LIN {X 0,Y 151.529,Z 477.279,A -85,B 0,C 180,E1 -25557.343,E2 -25557.343} C_VEL
LIN {X 0,Y 150.599,Z 472.699,A -85,B 0,C 180,E1 -25562.676,E2 -25562.676} C_VEL
LIN {X 0,Y 149.916,Z 471.492,A -85,B 0,C 180,E1 -25565.381,E2 -25565.381} C_VEL
LIN {X 0,Y 149.133,Z 469.93,A -85,B 0,C 180,E1 -25570.866,E2 -25570.866} C_VEL
LIN {X 0,Y 149.034,Z 469.641,A -85,B 0,C 180,E1 -25573.639,E2 -25573.639} C_VEL
LIN {X 0,Y 149.005,Z 470.056,A -85,B 0,C 180,E1 -25576.44,E2 -25576.44} C_VEL
LIN {X 0,Y 149.38,Z 472.272,A -85,B 0,C 180,E1 -25582.111,E2 -25582.111} C_VEL
LIN {X 0,Y 149.964,Z 473.797,A -85,B 0,C 180,E1 -25584.948,E2 -25584.948} C_VEL
LIN {X 0,Y 150.935,Z 477.352,A -85,B 0,C 180,E1 -25589.27,E2 -25589.27} C_VEL
LIN {X 0,Y 151.532,Z 479.613,A -85,B 0,C 180,E1 -25591.547,E2 -25591.547} C_VEL
LIN {X 0,Y 152.656,Z 484.991,A -85,B 0,C 180,E1 -25595.944,E2 -25595.944} C_VEL
LIN {X 0,Y 153.443,Z 490.683,A -85,B 0,C 180,E1 -25599.885,E2 -25599.885} C_VEL
LIN {X 0,Y 153.625,Z 494.117,A -85,B 0,C 180,E1 -25601.988,E2 -25601.988} C_VEL
LIN {X 0,Y 152.709,Z 497.182,A -85,B 0,C 180,E1 -25603.334,E2 -25603.334} C_VEL
LIN {X 0,Y 149.614,Z 504.051,A -85,B 0,C 180,E1 -25606.152,E2 -25606.152} C_VEL
LIN {X 0,Y 146.245,Z 509.783,A -85,B 0,C 180,E1 -25608.65,E2 -25608.65} C_VEL
LIN {X 0,Y 140.136,Z 517.083,A -85,B 0,C 180,E1 -25612.104,E2 -25612.104} C_VEL
LIN {X 0,Y 135.586,Z 522.016,A -85,B 0,C 180,E1 -25615.246,E2 -25615.246} C_VEL
LIN {X 0,Y 131.411,Z 526.277,A -85,B 0,C 180,E1 -25618.839,E2 -25618.839} C_VEL
LIN {X 0,Y 126.94,Z 530.452,A -85,B 0,C 180,E1 -25623.718,E2 -25623.718} C_VEL
LIN {X 0,Y 124.745,Z 532.341,A -85,B 0,C 180,E1 -25626.782,E2 -25626.782} C_VEL
LIN {X 0,Y 121.383,Z 534.797,A -85,B 0,C 180,E1 -25633.18,E2 -25633.18} C_VEL
LIN {X 0,Y 120.414,Z 535.442,A -85,B 0,C 180,E1 -25636.507,E2 -25636.507} C_VEL
LIN {X 0,Y 119.614,Z 535.472,A -85,B 0,C 180,E1 -25643.259,E2 -25643.259} C_VEL
LIN {X 0,Y 119.817,Z 535.003,A -85,B 0,C 180,E1 -25646.455,E2 -25646.455} C_VEL
LIN {X 0,Y 119.872,Z 537.944,A -85,B 0,C 180,E1 -25650.007,E2 -25650.007} C_VEL
LIN {X 0,Y 119.642,Z 540.145,A -85,B 0,C 180,E1 -25653.375,E2 -25653.375} C_VEL
LIN {X 0,Y 119.954,Z 543.316,A -85,B 0,C 180,E1 -25660.131,E2 -25660.131} C_VEL
LIN {X 0,Y 121.791,Z 545.048,A -85,B 0,C 180,E1 -25666.777,E2 -25666.777} C_VEL
LIN {X 0,Y 125.299,Z 545.373,A -85,B 0,C 180,E1 -25673.125,E2 -25673.125} C_VEL
LIN {X 0,Y 130.477,Z 544.334,A -85,B 0,C 180,E1 -25679.005,E2 -25679.005} C_VEL
LIN {X 0,Y 137.027,Z 541.96,A -85,B 0,C 180,E1 -25684.352,E2 -25684.352} C_VEL
LIN {X 0,Y 141.958,Z 539.578,A -85,B 0,C 180,E1 -25687.614,E2 -25687.614} C_VEL
LIN {X 0,Y 148.919,Z 535.676,A -85,B 0,C 180,E1 -25691.361,E2 -25691.361} C_VEL
LIN {X 0,Y 158.387,Z 529.476,A -85,B 0,C 180,E1 -25695.238,E2 -25695.238} C_VEL
LIN {X 0,Y 168.495,Z 521.385,A -85,B 0,C 180,E1 -25698.665,E2 -25698.665} C_VEL
LIN {X 0,Y 172.952,Z 516.993,A -85,B 0,C 180,E1 -25700.547,E2 -25700.547} C_VEL
LIN {X 0,Y 173.856,Z 515.604,A -85,B 0,C 180,E1 -25701.553,E2 -25701.553} C_VEL
LIN {X 0,Y 174.199,Z 514.027,A -85,B 0,C 180,E1 -25703.8,E2 -25703.8} C_VEL
LIN {X 0,Y 174.325,Z 513.097,A -85,B 0,C 180,E1 -25705.637,E2 -25705.637} C_VEL
LIN {X 0,Y 174.233,Z 512.255,A -85,B 0,C 180,E1 -25708.373,E2 -25708.373} C_VEL
LIN {X 0,Y 174.071,Z 511.974,A -85,B 0,C 180,E1 -25711.02,E2 -25711.02} C_VEL
LIN {X 0,Y 173.707,Z 512.343,A -85,B 0,C 180,E1 -25713.573,E2 -25713.573} C_VEL
LIN {X 0,Y 173.276,Z 513.059,A -85,B 0,C 180,E1 -25716.071,E2 -25716.071} C_VEL
LIN {X 0,Y 172.771,Z 514.258,A -85,B 0,C 180,E1 -25718.524,E2 -25718.524} C_VEL
LIN {X 0,Y 171.874,Z 515.921,A -85,B 0,C 180,E1 -25720.905,E2 -25720.905} C_VEL
LIN {X 0,Y 171.363,Z 516.563,A -85,B 0,C 180,E1 -25721.435,E2 -25721.435} C_VEL
LIN {X 0,Y 169.769,Z 518.268,A -85,B 0,C 180,E1 -25722.476,E2 -25722.476} C_VEL
LIN {X 0,Y 166.792,Z 520.759,A -85,B 0,C 180,E1 -25723.488,E2 -25723.488} C_VEL
LIN {X 0,Y 161.612,Z 524.398,A -85,B 0,C 180,E1 -25724.542,E2 -25724.542} C_VEL
LIN {X 0,Y 153.298,Z 529.29,A -85,B 0,C 180,E1 -25726.014,E2 -25726.014} C_VEL
LIN {X 0,Y 148.832,Z 531.676,A -85,B 0,C 180,E1 -25727.35,E2 -25727.35} C_VEL
LIN {X 0,Y 140.244,Z 535.91,A -85,B 0,C 180,E1 -25731.353,E2 -25731.353} C_VEL
LIN {X 0,Y 134.065,Z 538.329,A -85,B 0,C 180,E1 -25734.95,E2 -25734.95} C_VEL
LIN {X 0,Y 126.522,Z 540.322,A -85,B 0,C 180,E1 -25740.518,E2 -25740.518} C_VEL
LIN {X 0,Y 120.343,Z 540.847,A -85,B 0,C 180,E1 -25746.83,E2 -25746.83} C_VEL
LIN {X 0,Y 115.797,Z 539.767,A -85,B 0,C 180,E1 -25753.787,E2 -25753.787} C_VEL
LIN {X 0,Y 113.961,Z 538.469,A -85,B 0,C 180,E1 -25757.959,E2 -25757.959} C_VEL
LIN {X 0,Y 112.333,Z 535.676,A -85,B 0,C 180,E1 -25763.994,E2 -25763.994} C_VEL
LIN {X 0,Y 111.841,Z 531.696,A -85,B 0,C 180,E1 -25770.178,E2 -25770.178} C_VEL
LIN {X 0,Y 112.339,Z 525.917,A -85,B 0,C 180,E1 -25776.849,E2 -25776.849} C_VEL
LIN {X 0,Y 113.501,Z 518.907,A -85,B 0,C 180,E1 -25782.93,E2 -25782.93} C_VEL
LIN {X 0,Y 115.177,Z 510.671,A -85,B 0,C 180,E1 -25788.463,E2 -25788.463} C_VEL
LIN {X 0,Y 117.303,Z 501.805,A -85,B 0,C 180,E1 -25793.184,E2 -25793.184} C_VEL
LIN {X 0,Y 119.839,Z 492.117,A -85,B 0,C 180,E1 -25797.253,E2 -25797.253} C_VEL
LIN {X 0,Y 122.604,Z 481.332,A -85,B 0,C 180,E1 -25800.833,E2 -25800.833} C_VEL
LIN {X 0,Y 122.742,Z 478.141,A -85,B 0,C 180,E1 -25801.804,E2 -25801.804} C_VEL
LIN {X 0,Y 121.803,Z 465.816,A -85,B 0,C 180,E1 -25805.264,E2 -25805.264} C_VEL
LIN {X 0,Y 120.441,Z 453.323,A -85,B 0,C 180,E1 -25808.154,E2 -25808.154} C_VEL
LIN {X 0,Y 118.531,Z 439.707,A -85,B 0,C 180,E1 -25810.735,E2 -25810.735} C_VEL
LIN {X 0,Y 116.291,Z 431.963,A -85,B 0,C 180,E1 -25812.177,E2 -25812.177} C_VEL
LIN {X 0,Y 116.052,Z 430.282,A -85,B 0,C 180,E1 -25814.359,E2 -25814.359} C_VEL
LIN {X 0,Y 116.35,Z 432.329,A -85,B 0,C 180,E1 -25818.395,E2 -25818.395} C_VEL
LIN {X 0,Y 117.698,Z 435.529,A -85,B 0,C 180,E1 -25819.287,E2 -25819.287} C_VEL
LIN {X 0,Y 120.282,Z 441.063,A -85,B 0,C 180,E1 -25820.954,E2 -25820.954} C_VEL
LIN {X 0,Y 122.657,Z 447.493,A -85,B 0,C 180,E1 -25822.837,E2 -25822.837} C_VEL
LIN {X 0,Y 124.295,Z 458.548,A -85,B 0,C 180,E1 -25825.764,E2 -25825.764} C_VEL
LIN {X 0,Y 125.077,Z 468.612,A -85,B 0,C 180,E1 -25828.786,E2 -25828.786} C_VEL
LIN {X 0,Y 125.196,Z 477.893,A -85,B 0,C 180,E1 -25832.003,E2 -25832.003} C_VEL
LIN {X 0,Y 124.883,Z 480.197,A -85,B 0,C 180,E1 -25832.815,E2 -25832.815} C_VEL
LIN {X 0,Y 121.592,Z 490.126,A -85,B 0,C 180,E1 -25836.631,E2 -25836.631} C_VEL
LIN {X 0,Y 119.093,Z 497.329,A -85,B 0,C 180,E1 -25840.189,E2 -25840.189} C_VEL
LIN {X 0,Y 116.442,Z 504.956,A -85,B 0,C 180,E1 -25845.055,E2 -25845.055} C_VEL
LIN {X 0,Y 114.536,Z 510.57,A -85,B 0,C 180,E1 -25849.715,E2 -25849.715} C_VEL
LIN {X 0,Y 113.385,Z 514.456,A -85,B 0,C 180,E1 -25853.825,E2 -25853.825} C_VEL
LIN {X 0,Y 112.444,Z 518.81,A -85,B 0,C 180,E1 -25859.991,E2 -25859.991} C_VEL
LIN {X 0,Y 112.492,Z 521.446,A -85,B 0,C 180,E1 -25865.692,E2 -25865.692} C_VEL
LIN {X 0,Y 113.734,Z 523.058,A -85,B 0,C 180,E1 -25872.141,E2 -25872.141} C_VEL
LIN {X 0,Y 116.127,Z 523.197,A -85,B 0,C 180,E1 -25878.264,E2 -25878.264} C_VEL
LIN {X 0,Y 119.548,Z 522.01,A -85,B 0,C 180,E1 -25883.995,E2 -25883.995} C_VEL
LIN {X 0,Y 123.861,Z 519.524,A -85,B 0,C 180,E1 -25889.293,E2 -25889.293} C_VEL
LIN {X 0,Y 129.15,Z 515.615,A -85,B 0,C 180,E1 -25894.194,E2 -25894.194} C_VEL
LIN {X 0,Y 135.374,Z 510.135,A -85,B 0,C 180,E1 -25898.691,E2 -25898.691} C_VEL
LIN {X 0,Y 141.918,Z 503.34,A -85,B 0,C 180,E1 -25902.512,E2 -25902.512} C_VEL
LIN {X 0,Y 143.832,Z 500.919,A -85,B 0,C 180,E1 -25903.684,E2 -25903.684} C_VEL
LIN {X 0,Y 146.29,Z 494.851,A -85,B 0,C 180,E1 -25907.516,E2 -25907.516} C_VEL
LIN {X 0,Y 146.935,Z 492.599,A -85,B 0,C 180,E1 -25908.971,E2 -25908.971} C_VEL
LIN {X 0,Y 147.317,Z 488.968,A -85,B 0,C 180,E1 -25911.773,E2 -25911.773} C_VEL
LIN {X 0,Y 147.181,Z 484.415,A -85,B 0,C 180,E1 -25915.894,E2 -25915.894} C_VEL
LIN {X 0,Y 146.782,Z 480.742,A -85,B 0,C 180,E1 -25920.001,E2 -25920.001} C_VEL
LIN {X 0,Y 146.527,Z 478.659,A -85,B 0,C 180,E1 -25922.75,E2 -25922.75} C_VEL
LIN {X 0,Y 146.034,Z 477.435,A -85,B 0,C 180,E1 -25925.524,E2 -25925.524} C_VEL
LIN {X 0,Y 145.436,Z 475.978,A -85,B 0,C 180,E1 -25931.146,E2 -25931.146} C_VEL
LIN {X 0,Y 145.33,Z 475.906,A -85,B 0,C 180,E1 -25934.749,E2 -25934.749} C_VEL
LIN {X 0,Y 145.328,Z 476.304,A -85,B 0,C 180,E1 -25936.868,E2 -25936.868} C_VEL
LIN {X 0,Y 145.689,Z 478.652,A -85,B 0,C 180,E1 -25942.702,E2 -25942.702} C_VEL
LIN {X 0,Y 146.427,Z 481.664,A -85,B 0,C 180,E1 -25947.395,E2 -25947.395} C_VEL
LIN {X 0,Y 147.127,Z 485.666,A -85,B 0,C 180,E1 -25951.7,E2 -25951.7} C_VEL
LIN {X 0,Y 147.798,Z 490.757,A -85,B 0,C 180,E1 -25956.075,E2 -25956.075} C_VEL
LIN {X 0,Y 148.079,Z 495.842,A -85,B 0,C 180,E1 -25959.813,E2 -25959.813} C_VEL
LIN {X 0,Y 148.088,Z 497.025,A -85,B 0,C 180,E1 -25960.606,E2 -25960.606} C_VEL
LIN {X 0,Y 147.753,Z 498.436,A -85,B 0,C 180,E1 -25961.375,E2 -25961.375} C_VEL
LIN {X 0,Y 143.692,Z 506.293,A -85,B 0,C 180,E1 -25964.841,E2 -25964.841} C_VEL
LIN {X 0,Y 140.994,Z 510.362,A -85,B 0,C 180,E1 -25966.744,E2 -25966.744} C_VEL
LIN {X 0,Y 134.628,Z 517.484,A -85,B 0,C 180,E1 -25970.256,E2 -25970.256} C_VEL
LIN {X 0,Y 129.804,Z 522.272,A -85,B 0,C 180,E1 -25973.456,E2 -25973.456} C_VEL
LIN {X 0,Y 125.025,Z 526.714,A -85,B 0,C 180,E1 -25977.481,E2 -25977.481} C_VEL
LIN {X 0,Y 120.602,Z 530.421,A -85,B 0,C 180,E1 -25982.221,E2 -25982.221} C_VEL
LIN {X 0,Y 116.168,Z 533.546,A -85,B 0,C 180,E1 -25988.725,E2 -25988.725} C_VEL
LIN {X 0,Y 114.561,Z 534.519,A -85,B 0,C 180,E1 -25992.146,E2 -25992.146} C_VEL
LIN {X 0,Y 112.803,Z 535.205,A -85,B 0,C 180,E1 -25999.236,E2 -25999.236} C_VEL
LIN {X 0,Y 112.708,Z 534.402,A -85,B 0,C 180,E1 -26006.122,E2 -26006.122} C_VEL
LIN {X 0,Y 112.783,Z 534.396,A -85,B 0,C 180,E1 -26006.972,E2 -26006.972} C_VEL
LIN {X 0,Y 112.834,Z 536.832,A -85,B 0,C 180,E1 -26010.008,E2 -26010.008} C_VEL
LIN {X 0,Y 112.625,Z 539.19,A -85,B 0,C 180,E1 -26013.586,E2 -26013.586} C_VEL
LIN {X 0,Y 112.632,Z 541.123,A -85,B 0,C 180,E1 -26017.177,E2 -26017.177} C_VEL
LIN {X 0,Y 113.776,Z 543.763,A -85,B 0,C 180,E1 -26024.313,E2 -26024.313} C_VEL
LIN {X 0,Y 116.617,Z 545.034,A -85,B 0,C 180,E1 -26031.206,E2 -26031.206} C_VEL
LIN {X 0,Y 121.373,Z 544.981,A -85,B 0,C 180,E1 -26037.603,E2 -26037.603} C_VEL
LIN {X 0,Y 127.623,Z 543.547,A -85,B 0,C 180,E1 -26043.421,E2 -26043.421} C_VEL
LIN {X 0,Y 136.006,Z 540.379,A -85,B 0,C 180,E1 -26049.183,E2 -26049.183} C_VEL
LIN {X 0,Y 143.72,Z 536.597,A -85,B 0,C 180,E1 -26053.212,E2 -26053.212} C_VEL
LIN {X 0,Y 153.547,Z 530.753,A -85,B 0,C 180,E1 -26057.089,E2 -26057.089} C_VEL
LIN {X 0,Y 162.753,Z 524.224,A -85,B 0,C 180,E1 -26060.046,E2 -26060.046} C_VEL
LIN {X 0,Y 166.384,Z 521.137,A -85,B 0,C 180,E1 -26061.399,E2 -26061.399} C_VEL
LIN {X 0,Y 168.244,Z 519.215,A -85,B 0,C 180,E1 -26062.538,E2 -26062.538} C_VEL
LIN {X 0,Y 168.602,Z 518.152,A -85,B 0,C 180,E1 -26064.297,E2 -26064.297} C_VEL
LIN {X 0,Y 168.689,Z 517.021,A -85,B 0,C 180,E1 -26067.206,E2 -26067.206} C_VEL
LIN {X 0,Y 168.537,Z 516.48,A -85,B 0,C 180,E1 -26071.137,E2 -26071.137} C_VEL
LIN {X 0,Y 168.324,Z 516.604,A -85,B 0,C 180,E1 -26072.658,E2 -26072.658} C_VEL
LIN {X 0,Y 167.803,Z 517.219,A -85,B 0,C 180,E1 -26075.239,E2 -26075.239} C_VEL
LIN {X 0,Y 167.189,Z 518.231,A -85,B 0,C 180,E1 -26077.769,E2 -26077.769} C_VEL
LIN {X 0,Y 166.06,Z 519.805,A -85,B 0,C 180,E1 -26080.266,E2 -26080.266} C_VEL
LIN {X 0,Y 164.796,Z 521.052,A -85,B 0,C 180,E1 -26081.345,E2 -26081.345} C_VEL
LIN {X 0,Y 162.058,Z 523.259,A -85,B 0,C 180,E1 -26082.583,E2 -26082.583} C_VEL
LIN {X 0,Y 152.787,Z 529.415,A -85,B 0,C 180,E1 -26085.783,E2 -26085.783} C_VEL
LIN {X 0,Y 148.832,Z 531.676,A -85,B 0,C 180,E1 -26087.35,E2 -26087.35} C_VEL
LIN {X 0,Y 144.658,Z 533.752,A -85,B 0,C 180,E1 -26088.777,E2 -26088.777} C_VEL
LIN {X 0,Y 136.706,Z 536.782,A -85,B 0,C 180,E1 -26090.863,E2 -26090.863} C_VEL
LIN {X 0,Y 128.926,Z 539.051,A -85,B 0,C 180,E1 -26093.295,E2 -26093.295} C_VEL
LIN {X 0,Y 125.129,Z 539.915,A -85,B 0,C 180,E1 -26095.275,E2 -26095.275} C_VEL
LIN {X 0,Y 119.118,Z 540.944,A -85,B 0,C 180,E1 -26099.999,E2 -26099.999} C_VEL
LIN {X 0,Y 113.149,Z 540.911,A -85,B 0,C 180,E1 -26106.322,E2 -26106.322} C_VEL
LIN {X 0,Y 108.517,Z 539.326,A -85,B 0,C 180,E1 -26113.693,E2 -26113.693} C_VEL
LIN {X 0,Y 105.741,Z 536.232,A -85,B 0,C 180,E1 -26121.468,E2 -26121.468} C_VEL
LIN {X 0,Y 104.828,Z 532.437,A -85,B 0,C 180,E1 -26127.988,E2 -26127.988} C_VEL
LIN {X 0,Y 104.98,Z 527.294,A -85,B 0,C 180,E1 -26134.597,E2 -26134.597} C_VEL
LIN {X 0,Y 105.833,Z 521.559,A -85,B 0,C 180,E1 -26140.349,E2 -26140.349} C_VEL
LIN {X 0,Y 107.241,Z 514.282,A -85,B 0,C 180,E1 -26146.126,E2 -26146.126} C_VEL
LIN {X 0,Y 109.169,Z 506.012,A -85,B 0,C 180,E1 -26151.311,E2 -26151.311} C_VEL
LIN {X 0,Y 111.844,Z 495.677,A -85,B 0,C 180,E1 -26156.361,E2 -26156.361} C_VEL
LIN {X 0,Y 114.506,Z 485.811,A -85,B 0,C 180,E1 -26160.149,E2 -26160.149} C_VEL
LIN {X 0,Y 115.847,Z 480.256,A -85,B 0,C 180,E1 -26161.947,E2 -26161.947} C_VEL
LIN {X 0,Y 115.051,Z 467.836,A -85,B 0,C 180,E1 -26165.737,E2 -26165.737} C_VEL
LIN {X 0,Y 113.913,Z 456.148,A -85,B 0,C 180,E1 -26168.74,E2 -26168.74} C_VEL
LIN {X 0,Y 112.319,Z 443.599,A -85,B 0,C 180,E1 -26171.406,E2 -26171.406} C_VEL
LIN {X 0,Y 111.216,Z 438.554,A -85,B 0,C 180,E1 -26172.407,E2 -26172.407} C_VEL
LIN {X 0,Y 109.141,Z 432.087,A -85,B 0,C 180,E1 -26173.749,E2 -26173.749} C_VEL
LIN {X 0,Y 109.128,Z 431.825,A -85,B 0,C 180,E1 -26174.371,E2 -26174.371} C_VEL
LIN {X 0,Y 109.187,Z 432.383,A -85,B 0,C 180,E1 -26175.655,E2 -26175.655} C_VEL
LIN {X 0,Y 110.65,Z 435.876,A -85,B 0,C 180,E1 -26176.757,E2 -26176.757} C_VEL
LIN {X 0,Y 114.561,Z 444.315,A -85,B 0,C 180,E1 -26179.659,E2 -26179.659} C_VEL
LIN {X 0,Y 116.577,Z 449.72,A -85,B 0,C 180,E1 -26181.435,E2 -26181.435} C_VEL
LIN {X 0,Y 118.069,Z 461.172,A -85,B 0,C 180,E1 -26184.745,E2 -26184.745} C_VEL
LIN {X 0,Y 118.572,Z 470.679,A -85,B 0,C 180,E1 -26187.87,E2 -26187.87} C_VEL
LIN {X 0,Y 118.495,Z 479.723,A -85,B 0,C 180,E1 -26191.267,E2 -26191.267} C_VEL
LIN {X 0,Y 115.477,Z 488.788,A -85,B 0,C 180,E1 -26194.792,E2 -26194.792} C_VEL
LIN {X 0,Y 112.377,Z 497.254,A -85,B 0,C 180,E1 -26199.064,E2 -26199.064} C_VEL
LIN {X 0,Y 109.686,Z 504.599,A -85,B 0,C 180,E1 -26203.894,E2 -26203.894} C_VEL
LIN {X 0,Y 107.55,Z 510.582,A -85,B 0,C 180,E1 -26209.061,E2 -26209.061} C_VEL
LIN {X 0,Y 106.36,Z 514.469,A -85,B 0,C 180,E1 -26213.348,E2 -26213.348} C_VEL
LIN {X 0,Y 105.371,Z 518.896,A -85,B 0,C 180,E1 -26219.882,E2 -26219.882} C_VEL
LIN {X 0,Y 105.522,Z 521.986,A -85,B 0,C 180,E1 -26226.946,E2 -26226.946} C_VEL
LIN {X 0,Y 107.056,Z 523.532,A -85,B 0,C 180,E1 -26233.771,E2 -26233.771} C_VEL
LIN {X 0,Y 109.834,Z 523.597,A -85,B 0,C 180,E1 -26240.219,E2 -26240.219} C_VEL
LIN {X 0,Y 113.671,Z 522.362,A -85,B 0,C 180,E1 -26246.191,E2 -26246.191} C_VEL
LIN {X 0,Y 119.035,Z 519.417,A -85,B 0,C 180,E1 -26252.309,E2 -26252.309} C_VEL
LIN {X 0,Y 124.223,Z 515.867,A -85,B 0,C 180,E1 -26256.671,E2 -26256.671} C_VEL
LIN {X 0,Y 129.338,Z 511.713,A -85,B 0,C 180,E1 -26260.238,E2 -26260.238} C_VEL
LIN {X 0,Y 135.408,Z 506.028,A -85,B 0,C 180,E1 -26263.751,E2 -26263.751} C_VEL
LIN {X 0,Y 138.214,Z 502.999,A -85,B 0,C 180,E1 -26265.272,E2 -26265.272} C_VEL
LIN {X 0,Y 140.524,Z 498.388,A -85,B 0,C 180,E1 -26268.461,E2 -26268.461} C_VEL
LIN {X 0,Y 141.385,Z 496.228,A -85,B 0,C 180,E1 -26269.982,E2 -26269.982} C_VEL
LIN {X 0,Y 141.912,Z 493.778,A -85,B 0,C 180,E1 -26272.029,E2 -26272.029} C_VEL
LIN {X 0,Y 142.193,Z 489.948,A -85,B 0,C 180,E1 -26275.749,E2 -26275.749} C_VEL
LIN {X 0,Y 142.161,Z 486.348,A -85,B 0,C 180,E1 -26280.001,E2 -26280.001} C_VEL
LIN {X 0,Y 142.13,Z 484.381,A -85,B 0,C 180,E1 -26282.835,E2 -26282.835} C_VEL
LIN {X 0,Y 141.595,Z 482.751,A -85,B 0,C 180,E1 -26286.995,E2 -26286.995} C_VEL
LIN {X 0,Y 141.409,Z 481.81,A -85,B 0,C 180,E1 -26291.468,E2 -26291.468} C_VEL
LIN {X 0,Y 141.361,Z 481.741,A -85,B 0,C 180,E1 -26294.395,E2 -26294.395} C_VEL
LIN {X 0,Y 141.279,Z 482.935,A -85,B 0,C 180,E1 -26299.086,E2 -26299.086} C_VEL
LIN {X 0,Y 141.588,Z 484.8,A -85,B 0,C 180,E1 -26303.398,E2 -26303.398} C_VEL
LIN {X 0,Y 142.058,Z 487.938,A -85,B 0,C 180,E1 -26308.033,E2 -26308.033} C_VEL
LIN {X 0,Y 142.342,Z 491.327,A -85,B 0,C 180,E1 -26311.771,E2 -26311.771} C_VEL
LIN {X 0,Y 142.603,Z 496.26,A -85,B 0,C 180,E1 -26316.258,E2 -26316.258} C_VEL
LIN {X 0,Y 142.491,Z 499.587,A -85,B 0,C 180,E1 -26318.918,E2 -26318.918} C_VEL
LIN {X 0,Y 142.149,Z 501.244,A -85,B 0,C 180,E1 -26319.997,E2 -26319.997} C_VEL
LIN {X 0,Y 137.822,Z 508.431,A -85,B 0,C 180,E1 -26323.404,E2 -26323.404} C_VEL
LIN {X 0,Y 134.787,Z 512.255,A -85,B 0,C 180,E1 -26325.269,E2 -26325.269} C_VEL
LIN {X 0,Y 128.19,Z 518.864,A -85,B 0,C 180,E1 -26328.871,E2 -26328.871} C_VEL
LIN {X 0,Y 122.312,Z 524.12,A -85,B 0,C 180,E1 -26332.902,E2 -26332.902} C_VEL
LIN {X 0,Y 117.315,Z 528.221,A -85,B 0,C 180,E1 -26337.383,E2 -26337.383} C_VEL
LIN {X 0,Y 114.358,Z 530.351,A -85,B 0,C 180,E1 -26340.561,E2 -26340.561} C_VEL
LIN {X 0,Y 109.572,Z 533.346,A -85,B 0,C 180,E1 -26347.375,E2 -26347.375} C_VEL
LIN {X 0,Y 107.786,Z 534.204,A -85,B 0,C 180,E1 -26350.982,E2 -26350.982} C_VEL
LIN {X 0,Y 105.804,Z 534.762,A -85,B 0,C 180,E1 -26358.514,E2 -26358.514} C_VEL
LIN {X 0,Y 105.479,Z 534.445,A -85,B 0,C 180,E1 -26362.351,E2 -26362.351} C_VEL
LIN {X 0,Y 105.761,Z 533.557,A -85,B 0,C 180,E1 -26367.265,E2 -26367.265} C_VEL
LIN {X 0,Y 105.797,Z 535.71,A -85,B 0,C 180,E1 -26370.008,E2 -26370.008} C_VEL
LIN {X 0,Y 105.557,Z 539.233,A -85,B 0,C 180,E1 -26375.74,E2 -26375.74} C_VEL
LIN {X 0,Y 106.052,Z 541.831,A -85,B 0,C 180,E1 -26381.476,E2 -26381.476} C_VEL
LIN {X 0,Y 108.263,Z 544.074,A -85,B 0,C 180,E1 -26388.948,E2 -26388.948} C_VEL
LIN {X 0,Y 112.368,Z 544.916,A -85,B 0,C 180,E1 -26395.973,E2 -26395.973} C_VEL
LIN {X 0,Y 118.241,Z 544.445,A -85,B 0,C 180,E1 -26402.348,E2 -26402.348} C_VEL
LIN {X 0,Y 125.565,Z 542.674,A -85,B 0,C 180,E1 -26408.009,E2 -26408.009} C_VEL
LIN {X 0,Y 134.05,Z 539.522,A -85,B 0,C 180,E1 -26412.974,E2 -26412.974} C_VEL
LIN {X 0,Y 141.192,Z 536.241,A -85,B 0,C 180,E1 -26416.207,E2 -26416.207} C_VEL
LIN {X 0,Y 148.881,Z 532.042,A -85,B 0,C 180,E1 -26419.058,E2 -26419.058} C_VEL
LIN {X 0,Y 157.008,Z 526.843,A -85,B 0,C 180,E1 -26421.574,E2 -26421.574} C_VEL
LIN {X 0,Y 159.744,Z 524.894,A -85,B 0,C 180,E1 -26422.372,E2 -26422.372} C_VEL
LIN {X 0,Y 162.108,Z 523.059,A -85,B 0,C 180,E1 -26423.333,E2 -26423.333} C_VEL
LIN {X 0,Y 162.805,Z 521.914,A -85,B 0,C 180,E1 -26425.112,E2 -26425.112} C_VEL
LIN {X 0,Y 162.832,Z 520.793,A -85,B 0,C 180,E1 -26429.688,E2 -26429.688} C_VEL
LIN {X 0,Y 162.711,Z 520.674,A -85,B 0,C 180,E1 -26431.632,E2 -26431.632} C_VEL
LIN {X 0,Y 161.747,Z 521.583,A -85,B 0,C 180,E1 -26435.858,E2 -26435.858} C_VEL
LIN {X 0,Y 161.458,Z 521.946,A -85,B 0,C 180,E1 -26436.935,E2 -26436.935} C_VEL
LIN {X 0,Y 160.202,Z 523.33,A -85,B 0,C 180,E1 -26439.453,E2 -26439.453} C_VEL
LIN {X 0,Y 158.549,Z 524.61,A -85,B 0,C 180,E1 -26440.395,E2 -26440.395} C_VEL
LIN {X 0,Y 147.971,Z 530.961,A -85,B 0,C 180,E1 -26443.891,E2 -26443.891} C_VEL
LIN {X 0,Y 140.207,Z 534.788,A -85,B 0,C 180,E1 -26446.963,E2 -26446.963} C_VEL
LIN {X 0,Y 132.339,Z 537.877,A -85,B 0,C 180,E1 -26450.832,E2 -26450.832} C_VEL
LIN {X 0,Y 125.129,Z 539.915,A -85,B 0,C 180,E1 -26455.275,E2 -26455.275} C_VEL
LIN {X 0,Y 121.462,Z 540.629,A -85,B 0,C 180,E1 -26457.406,E2 -26457.406} C_VEL
LIN {X 0,Y 114.318,Z 541.204,A -85,B 0,C 180,E1 -26460.735,E2 -26460.735} C_VEL
LIN {X 0,Y 107.639,Z 541.003,A -85,B 0,C 180,E1 -26464.506,E2 -26464.506} C_VEL
LIN {X 0,Y 104.831,Z 540.477,A -85,B 0,C 180,E1 -26467.289,E2 -26467.289} C_VEL
LIN {X 0,Y 101.254,Z 538.717,A -85,B 0,C 180,E1 -26473.623,E2 -26473.623} C_VEL
LIN {X 0,Y 98.534,Z 535.066,A -85,B 0,C 180,E1 -26481.971,E2 -26481.971} C_VEL
LIN {X 0,Y 97.791,Z 531.584,A -85,B 0,C 180,E1 -26487.847,E2 -26487.847} C_VEL
LIN {X 0,Y 97.994,Z 526.13,A -85,B 0,C 180,E1 -26495.01,E2 -26495.01} C_VEL
LIN {X 0,Y 98.889,Z 520.153,A -85,B 0,C 180,E1 -26501.099,E2 -26501.099} C_VEL
LIN {X 0,Y 100.451,Z 512.359,A -85,B 0,C 180,E1 -26507.346,E2 -26507.346} C_VEL
LIN {X 0,Y 102.583,Z 503.646,A -85,B 0,C 180,E1 -26512.851,E2 -26512.851} C_VEL
LIN {X 0,Y 105.278,Z 493.91,A -85,B 0,C 180,E1 -26517.711,E2 -26517.711} C_VEL
LIN {X 0,Y 108.458,Z 482.477,A -85,B 0,C 180,E1 -26522.081,E2 -26522.081} C_VEL
LIN {X 0,Y 108.845,Z 479.437,A -85,B 0,C 180,E1 -26523.121,E2 -26523.121} C_VEL
LIN {X 0,Y 108.089,Z 467.27,A -85,B 0,C 180,E1 -26527.03,E2 -26527.03} C_VEL
LIN {X 0,Y 106.938,Z 455.012,A -85,B 0,C 180,E1 -26530.309,E2 -26530.309} C_VEL
LIN {X 0,Y 105.326,Z 442.615,A -85,B 0,C 180,E1 -26533.057,E2 -26533.057} C_VEL
LIN {X 0,Y 103.826,Z 437.818,A -85,B 0,C 180,E1 -26534.169,E2 -26534.169} C_VEL
LIN {X 0,Y 105.109,Z 439.248,A -85,B 0,C 180,E1 -26535.034,E2 -26535.034} C_VEL
LIN {X 0,Y 108.674,Z 447.246,A -85,B 0,C 180,E1 -26538.102,E2 -26538.102} C_VEL
LIN {X 0,Y 110.693,Z 452.874,A -85,B 0,C 180,E1 -26540.2,E2 -26540.2} C_VEL
LIN {X 0,Y 111.808,Z 463.777,A -85,B 0,C 180,E1 -26543.677,E2 -26543.677} C_VEL
LIN {X 0,Y 112.085,Z 473.804,A -85,B 0,C 180,E1 -26547.297,E2 -26547.297} C_VEL
LIN {X 0,Y 111.866,Z 480.43,A -85,B 0,C 180,E1 -26549.992,E2 -26549.992} C_VEL
LIN {X 0,Y 108.678,Z 489.409,A -85,B 0,C 180,E1 -26553.699,E2 -26553.699} C_VEL
LIN {X 0,Y 105.181,Z 498.511,A -85,B 0,C 180,E1 -26558.638,E2 -26558.638} C_VEL
LIN {X 0,Y 102.631,Z 505.127,A -85,B 0,C 180,E1 -26563.372,E2 -26563.372} C_VEL
LIN {X 0,Y 100.224,Z 511.598,A -85,B 0,C 180,E1 -26569.446,E2 -26569.446} C_VEL
LIN {X 0,Y 98.832,Z 516.228,A -85,B 0,C 180,E1 -26575.245,E2 -26575.245} C_VEL
LIN {X 0,Y 98.209,Z 519.537,A -85,B 0,C 180,E1 -26580.827,E2 -26580.827} C_VEL
LIN {X 0,Y 98.613,Z 522.527,A -85,B 0,C 180,E1 -26588.379,E2 -26588.379} C_VEL
LIN {X 0,Y 100.495,Z 523.99,A -85,B 0,C 180,E1 -26595.628,E2 -26595.628} C_VEL
LIN {X 0,Y 103.646,Z 524.005,A -85,B 0,C 180,E1 -26602.393,E2 -26602.393} C_VEL
LIN {X 0,Y 107.925,Z 522.742,A -85,B 0,C 180,E1 -26608.605,E2 -26608.605} C_VEL
LIN {X 0,Y 113.119,Z 520.167,A -85,B 0,C 180,E1 -26614.222,E2 -26614.222} C_VEL
LIN {X 0,Y 119.929,Z 515.851,A -85,B 0,C 180,E1 -26619.63,E2 -26619.63} C_VEL
LIN {X 0,Y 126.773,Z 510.472,A -85,B 0,C 180,E1 -26623.909,E2 -26623.909} C_VEL
LIN {X 0,Y 132.751,Z 504.938,A -85,B 0,C 180,E1 -26627.064,E2 -26627.064} C_VEL
LIN {X 0,Y 135.386,Z 500.476,A -85,B 0,C 180,E1 -26630.458,E2 -26630.458} C_VEL
LIN {X 0,Y 136.349,Z 497.905,A -85,B 0,C 180,E1 -26632.702,E2 -26632.702} C_VEL
LIN {X 0,Y 137.023,Z 493.935,A -85,B 0,C 180,E1 -26637.061,E2 -26637.061} C_VEL
LIN {X 0,Y 137.224,Z 491.699,A -85,B 0,C 180,E1 -26640.001,E2 -26640.001} C_VEL
LIN {X 0,Y 137.387,Z 489.786,A -85,B 0,C 180,E1 -26642.933,E2 -26642.933} C_VEL
LIN {X 0,Y 137.248,Z 488.558,A -85,B 0,C 180,E1 -26645.879,E2 -26645.879} C_VEL
LIN {X 0,Y 137.005,Z 487.379,A -85,B 0,C 180,E1 -26651.842,E2 -26651.842} C_VEL
LIN {X 0,Y 136.965,Z 487.458,A -85,B 0,C 180,E1 -26654.867,E2 -26654.867} C_VEL
LIN {X 0,Y 136.862,Z 488.176,A -85,B 0,C 180,E1 -26657.946,E2 -26657.946} C_VEL
LIN {X 0,Y 136.96,Z 489.955,A -85,B 0,C 180,E1 -26662.554,E2 -26662.554} C_VEL
LIN {X 0,Y 137.159,Z 491.76,A -85,B 0,C 180,E1 -26665.821,E2 -26665.821} C_VEL
LIN {X 0,Y 137.254,Z 495.687,A -85,B 0,C 180,E1 -26670.801,E2 -26670.801} C_VEL
LIN {X 0,Y 137.064,Z 501.04,A -85,B 0,C 180,E1 -26676.133,E2 -26676.133} C_VEL
LIN {X 0,Y 136.74,Z 503.337,A -85,B 0,C 180,E1 -26678.081,E2 -26678.081} C_VEL
LIN {X 0,Y 134.883,Z 506.471,A -85,B 0,C 180,E1 -26679.789,E2 -26679.789} C_VEL
LIN {X 0,Y 131,Z 511.618,A -85,B 0,C 180,E1 -26682.478,E2 -26682.478} C_VEL
LIN {X 0,Y 125.22,Z 517.266,A -85,B 0,C 180,E1 -26685.459,E2 -26685.459} C_VEL
LIN {X 0,Y 118.701,Z 522.756,A -85,B 0,C 180,E1 -26689.373,E2 -26689.373} C_VEL
LIN {X 0,Y 112.407,Z 527.502,A -85,B 0,C 180,E1 -26694.372,E2 -26694.372} C_VEL
LIN {X 0,Y 108.219,Z 530.283,A -85,B 0,C 180,E1 -26698.709,E2 -26698.709} C_VEL
LIN {X 0,Y 105.397,Z 531.909,A -85,B 0,C 180,E1 -26702.186,E2 -26702.186} C_VEL
LIN {X 0,Y 103.018,Z 533.103,A -85,B 0,C 180,E1 -26705.848,E2 -26705.848} C_VEL
LIN {X 0,Y 99.699,Z 534.287,A -85,B 0,C 180,E1 -26713.632,E2 -26713.632} C_VEL
LIN {X 0,Y 98.834,Z 534.297,A -85,B 0,C 180,E1 -26717.692,E2 -26717.692} C_VEL
LIN {X 0,Y 98.609,Z 533.014,A -85,B 0,C 180,E1 -26726.223,E2 -26726.223} C_VEL
LIN {X 0,Y 98.738,Z 532.712,A -85,B 0,C 180,E1 -26727.759,E2 -26727.759} C_VEL
LIN {X 0,Y 98.698,Z 536.188,A -85,B 0,C 180,E1 -26732.671,E2 -26732.671} C_VEL
LIN {X 0,Y 98.666,Z 539.238,A -85,B 0,C 180,E1 -26738.199,E2 -26738.199} C_VEL
LIN {X 0,Y 100.106,Z 542.394,A -85,B 0,C 180,E1 -26746.318,E2 -26746.318} C_VEL
LIN {X 0,Y 103.488,Z 544.186,A -85,B 0,C 180,E1 -26754.055,E2 -26754.055} C_VEL
LIN {X 0,Y 108.953,Z 544.693,A -85,B 0,C 180,E1 -26761.076,E2 -26761.076} C_VEL
LIN {X 0,Y 116.054,Z 543.854,A -85,B 0,C 180,E1 -26767.279,E2 -26767.279} C_VEL
LIN {X 0,Y 124.349,Z 541.7,A -85,B 0,C 180,E1 -26772.713,E2 -26772.713} C_VEL
LIN {X 0,Y 133.823,Z 538.234,A -85,B 0,C 180,E1 -26777.336,E2 -26777.336} C_VEL
LIN {X 0,Y 144.384,Z 533.225,A -85,B 0,C 180,E1 -26781.16,E2 -26781.16} C_VEL
LIN {X 0,Y 155.623,Z 526.607,A -85,B 0,C 180,E1 -26784.387,E2 -26784.387} C_VEL
LIN {X 0,Y 156.807,Z 525.068,A -85,B 0,C 180,E1 -26787.463,E2 -26787.463} C_VEL
LIN {X 0,Y 156.833,Z 524.603,A -85,B 0,C 180,E1 -26790.466,E2 -26790.466} C_VEL
LIN {X 0,Y 156.153,Z 524.965,A -85,B 0,C 180,E1 -26794.187,E2 -26794.187} C_VEL
LIN {X 0,Y 155.626,Z 525.411,A -85,B 0,C 180,E1 -26796.018,E2 -26796.018} C_VEL
LIN {X 0,Y 153.828,Z 526.821,A -85,B 0,C 180,E1 -26798.561,E2 -26798.561} C_VEL
LIN {X 0,Y 143.367,Z 532.476,A -85,B 0,C 180,E1 -26801.847,E2 -26801.847} C_VEL
LIN {X 0,Y 135.188,Z 536.021,A -85,B 0,C 180,E1 -26804.933,E2 -26804.933} C_VEL
LIN {X 0,Y 129.594,Z 537.996,A -85,B 0,C 180,E1 -26807.489,E2 -26807.489} C_VEL
LIN {X 0,Y 120.49,Z 540.377,A -85,B 0,C 180,E1 -26812.607,E2 -26812.607} C_VEL
LIN {X 0,Y 112.491,Z 541.319,A -85,B 0,C 180,E1 -26818.682,E2 -26818.682} C_VEL
LIN {X 0,Y 105.96,Z 540.789,A -85,B 0,C 180,E1 -26825.718,E2 -26825.718} C_VEL
LIN {X 0,Y 104.831,Z 540.477,A -85,B 0,C 180,E1 -26827.289,E2 -26827.289} C_VEL
LIN {X 0,Y 102.295,Z 539.736,A -85,B 0,C 180,E1 -26830.212,E2 -26830.212} C_VEL
LIN {X 0,Y 97.053,Z 537.844,A -85,B 0,C 180,E1 -26834.927,E2 -26834.927} C_VEL
LIN {X 0,Y 93.245,Z 535.74,A -85,B 0,C 180,E1 -26838.957,E2 -26838.957} C_VEL
LIN {X 0,Y 91.45,Z 533.882,A -85,B 0,C 180,E1 -26842.276,E2 -26842.276} C_VEL
LIN {X 0,Y 91.175,Z 533.213,A -85,B 0,C 180,E1 -26843.435,E2 -26843.435} C_VEL
LIN {X 0,Y 90.727,Z 529.354,A -85,B 0,C 180,E1 -26849.598,E2 -26849.598} C_VEL
LIN {X 0,Y 91.186,Z 523.79,A -85,B 0,C 180,E1 -26856.676,E2 -26856.676} C_VEL
LIN {X 0,Y 92.282,Z 517.203,A -85,B 0,C 180,E1 -26863.267,E2 -26863.267} C_VEL
LIN {X 0,Y 94.154,Z 508.643,A -85,B 0,C 180,E1 -26869.913,E2 -26869.913} C_VEL
LIN {X 0,Y 96.739,Z 499.053,A -85,B 0,C 180,E1 -26875.723,E2 -26875.723} C_VEL
LIN {X 0,Y 99.598,Z 489.162,A -85,B 0,C 180,E1 -26880.39,E2 -26880.39} C_VEL
LIN {X 0,Y 101.602,Z 482.175,A -85,B 0,C 180,E1 -26883.053,E2 -26883.053} C_VEL
LIN {X 0,Y 101.867,Z 479.669,A -85,B 0,C 180,E1 -26883.973,E2 -26883.973} C_VEL
LIN {X 0,Y 101.225,Z 467.72,A -85,B 0,C 180,E1 -26888.079,E2 -26888.079} C_VEL
LIN {X 0,Y 100.16,Z 455.255,A -85,B 0,C 180,E1 -26891.672,E2 -26891.672} C_VEL
LIN {X 0,Y 99.191,Z 446.464,A -85,B 0,C 180,E1 -26893.887,E2 -26893.887} C_VEL
LIN {X 0,Y 100.134,Z 447.445,A -85,B 0,C 180,E1 -26894.568,E2 -26894.568} C_VEL
LIN {X 0,Y 101.683,Z 447.868,A -85,B 0,C 180,E1 -26895.378,E2 -26895.378} C_VEL
LIN {X 0,Y 102.789,Z 449.949,A -85,B 0,C 180,E1 -26896.387,E2 -26896.387} C_VEL
LIN {X 0,Y 104.835,Z 456.249,A -85,B 0,C 180,E1 -26898.926,E2 -26898.926} C_VEL
LIN {X 0,Y 105.578,Z 467.18,A -85,B 0,C 180,E1 -26902.822,E2 -26902.822} C_VEL
LIN {X 0,Y 105.544,Z 476.732,A -85,B 0,C 180,E1 -26906.651,E2 -26906.651} C_VEL
LIN {X 0,Y 105.285,Z 481.045,A -85,B 0,C 180,E1 -26908.557,E2 -26908.557} C_VEL
LIN {X 0,Y 102.341,Z 488.961,A -85,B 0,C 180,E1 -26911.959,E2 -26911.959} C_VEL
LIN {X 0,Y 98.572,Z 498.258,A -85,B 0,C 180,E1 -26917.195,E2 -26917.195} C_VEL
LIN {X 0,Y 95.58,Z 505.603,A -85,B 0,C 180,E1 -26922.734,E2 -26922.734} C_VEL
LIN {X 0,Y 92.922,Z 512.605,A -85,B 0,C 180,E1 -26929.887,E2 -26929.887} C_VEL
LIN {X 0,Y 91.404,Z 517.842,A -85,B 0,C 180,E1 -26937.462,E2 -26937.462} C_VEL
LIN {X 0,Y 91.071,Z 520.476,A -85,B 0,C 180,E1 -26942.684,E2 -26942.684} C_VEL
LIN {X 0,Y 91.801,Z 523.059,A -85,B 0,C 180,E1 -26950.045,E2 -26950.045} C_VEL
LIN {X 0,Y 94.228,Z 524.472,A -85,B 0,C 180,E1 -26958.216,E2 -26958.216} C_VEL
LIN {X 0,Y 97.665,Z 524.415,A -85,B 0,C 180,E1 -26964.854,E2 -26964.854} C_VEL
LIN {X 0,Y 102.441,Z 523.106,A -85,B 0,C 180,E1 -26971.301,E2 -26971.301} C_VEL
LIN {X 0,Y 108.179,Z 520.487,A -85,B 0,C 180,E1 -26977.059,E2 -26977.059} C_VEL
LIN {X 0,Y 115.122,Z 516.429,A -85,B 0,C 180,E1 -26982.229,E2 -26982.229} C_VEL
LIN {X 0,Y 122.924,Z 510.698,A -85,B 0,C 180,E1 -26986.781,E2 -26986.781} C_VEL
LIN {X 0,Y 127.119,Z 507.153,A -85,B 0,C 180,E1 -26988.845,E2 -26988.845} C_VEL
LIN {X 0,Y 128.792,Z 504.962,A -85,B 0,C 180,E1 -26990.579,E2 -26990.579} C_VEL
LIN {X 0,Y 130.069,Z 502.974,A -85,B 0,C 180,E1 -26992.238,E2 -26992.238} C_VEL
LIN {X 0,Y 130.768,Z 501.455,A -85,B 0,C 180,E1 -26993.831,E2 -26993.831} C_VEL
LIN {X 0,Y 131.755,Z 497.759,A -85,B 0,C 180,E1 -26998.473,E2 -26998.473} C_VEL
LIN {X 0,Y 132.326,Z 494.92,A -85,B 0,C 180,E1 -27003.046,E2 -27003.046} C_VEL
LIN {X 0,Y 132.389,Z 493.687,A -85,B 0,C 180,E1 -27006.096,E2 -27006.096} C_VEL
LIN {X 0,Y 132.307,Z 492.689,A -85,B 0,C 180,E1 -27012.268,E2 -27012.268} C_VEL
LIN {X 0,Y 132.147,Z 493.259,A -85,B 0,C 180,E1 -27016.832,E2 -27016.832} C_VEL
LIN {X 0,Y 132.097,Z 494.933,A -85,B 0,C 180,E1 -27021.866,E2 -27021.866} C_VEL
LIN {X 0,Y 132.138,Z 496.631,A -85,B 0,C 180,E1 -27025.306,E2 -27025.306} C_VEL
LIN {X 0,Y 131.979,Z 499.645,A -85,B 0,C 180,E1 -27029.561,E2 -27029.561} C_VEL
LIN {X 0,Y 131.52,Z 503.656,A -85,B 0,C 180,E1 -27034.132,E2 -27034.132} C_VEL
LIN {X 0,Y 131.101,Z 506.028,A -85,B 0,C 180,E1 -27036.489,E2 -27036.489} C_VEL
LIN {X 0,Y 130.605,Z 506.993,A -85,B 0,C 180,E1 -27037.147,E2 -27037.147} C_VEL
LIN {X 0,Y 126.301,Z 512.255,A -85,B 0,C 180,E1 -27040.095,E2 -27040.095} C_VEL
LIN {X 0,Y 120.28,Z 517.687,A -85,B 0,C 180,E1 -27043.094,E2 -27043.094} C_VEL
LIN {X 0,Y 113.399,Z 522.997,A -85,B 0,C 180,E1 -27047.033,E2 -27047.033} C_VEL
LIN {X 0,Y 106.259,Z 527.844,A -85,B 0,C 180,E1 -27052.534,E2 -27052.534} C_VEL
LIN {X 0,Y 102.207,Z 530.238,A -85,B 0,C 180,E1 -27056.638,E2 -27056.638} C_VEL
LIN {X 0,Y 99.139,Z 531.758,A -85,B 0,C 180,E1 -27060.26,E2 -27060.26} C_VEL
LIN {X 0,Y 94.405,Z 533.561,A -85,B 0,C 180,E1 -27068.158,E2 -27068.158} C_VEL
LIN {X 0,Y 92.877,Z 533.889,A -85,B 0,C 180,E1 -27072.392,E2 -27072.392} C_VEL
LIN {X 0,Y 91.409,Z 533.309,A -85,B 0,C 180,E1 -27081.165,E2 -27081.165} C_VEL
LIN {X 0,Y 91.767,Z 531.841,A -85,B 0,C 180,E1 -27088.331,E2 -27088.331} C_VEL
LIN {X 0,Y 91.752,Z 533.958,A -85,B 0,C 180,E1 -27091.311,E2 -27091.311} C_VEL
LIN {X 0,Y 91.71,Z 538.151,A -85,B 0,C 180,E1 -27098.826,E2 -27098.826} C_VEL
LIN {X 0,Y 93.333,Z 541.612,A -85,B 0,C 180,E1 -27107.539,E2 -27107.539} C_VEL
LIN {X 0,Y 97.044,Z 543.677,A -85,B 0,C 180,E1 -27115.765,E2 -27115.765} C_VEL
LIN {X 0,Y 102.925,Z 544.431,A -85,B 0,C 180,E1 -27123.12,E2 -27123.12} C_VEL
LIN {X 0,Y 110.483,Z 543.906,A -85,B 0,C 180,E1 -27129.512,E2 -27129.512} C_VEL
LIN {X 0,Y 119.253,Z 542.114,A -85,B 0,C 180,E1 -27135.017,E2 -27135.017} C_VEL
LIN {X 0,Y 129.146,Z 538.958,A -85,B 0,C 180,E1 -27139.638,E2 -27139.638} C_VEL
LIN {X 0,Y 140.091,Z 534.387,A -85,B 0,C 180,E1 -27143.396,E2 -27143.396} C_VEL
LIN {X 0,Y 148.756,Z 529.895,A -85,B 0,C 180,E1 -27145.779,E2 -27145.779} C_VEL
LIN {X 0,Y 150.384,Z 528.751,A -85,B 0,C 180,E1 -27147.276,E2 -27147.276} C_VEL
LIN {X 0,Y 150.68,Z 528.316,A -85,B 0,C 180,E1 -27149.131,E2 -27149.131} C_VEL
LIN {X 0,Y 150.216,Z 528.277,A -85,B 0,C 180,E1 -27152.749,E2 -27152.749} C_VEL
LIN {X 0,Y 149.632,Z 528.632,A -85,B 0,C 180,E1 -27154.993,E2 -27154.993} C_VEL
LIN {X 0,Y 148.797,Z 529.147,A -85,B 0,C 180,E1 -27156.329,E2 -27156.329} C_VEL
LIN {X 0,Y 146.36,Z 530.454,A -85,B 0,C 180,E1 -27157.408,E2 -27157.408} C_VEL
LIN {X 0,Y 136.581,Z 534.892,A -85,B 0,C 180,E1 -27160.459,E2 -27160.459} C_VEL
LIN {X 0,Y 127.41,Z 538.114,A -85,B 0,C 180,E1 -27163.989,E2 -27163.989} C_VEL
LIN {X 0,Y 121.778,Z 539.638,A -85,B 0,C 180,E1 -27166.652,E2 -27166.652} C_VEL
LIN {X 0,Y 113.798,Z 541.123,A -85,B 0,C 180,E1 -27171.209,E2 -27171.209} C_VEL
LIN {X 0,Y 105.528,Z 541.561,A -85,B 0,C 180,E1 -27177.564,E2 -27177.564} C_VEL
LIN {X 0,Y 98.786,Z 540.495,A -85,B 0,C 180,E1 -27185.032,E2 -27185.032} C_VEL
LIN {X 0,Y 93.987,Z 537.921,A -85,B 0,C 180,E1 -27193.534,E2 -27193.534} C_VEL
LIN {X 0,Y 91.824,Z 535.03,A -85,B 0,C 180,E1 -27200.091,E2 -27200.091} C_VEL
LIN {X 0,Y 91.175,Z 533.213,A -85,B 0,C 180,E1 -27203.435,E2 -27203.435} C_VEL
LIN {X 0,Y 90.149,Z 531.098,A -85,B 0,C 180,E1 -27206.84,E2 -27206.84} C_VEL
LIN {X 0,Y 88.491,Z 528.648,A -85,B 0,C 180,E1 -27210.143,E2 -27210.143} C_VEL
LIN {X 0,Y 84.943,Z 521.873,A -85,B 0,C 180,E1 -27217.907,E2 -27217.907} C_VEL
LIN {X 0,Y 84.797,Z 518.587,A -85,B 0,C 180,E1 -27221.302,E2 -27221.302} C_VEL
LIN {X 0,Y 86.49,Z 510.602,A -85,B 0,C 180,E1 -27228.442,E2 -27228.442} C_VEL
LIN {X 0,Y 88.998,Z 501.189,A -85,B 0,C 180,E1 -27234.958,E2 -27234.958} C_VEL
LIN {X 0,Y 92.001,Z 491.079,A -85,B 0,C 180,E1 -27240.333,E2 -27240.333} C_VEL
LIN {X 0,Y 94.811,Z 481.702,A -85,B 0,C 180,E1 -27244.219,E2 -27244.219} C_VEL
LIN {X 0,Y 94.619,Z 472.919,A -85,B 0,C 180,E1 -27247.615,E2 -27247.615} C_VEL
LIN {X 0,Y 93.918,Z 461.568,A -85,B 0,C 180,E1 -27251.446,E2 -27251.446} C_VEL
LIN {X 0,Y 93.405,Z 454.814,A -85,B 0,C 180,E1 -27253.43,E2 -27253.43} C_VEL
LIN {X 0,Y 94.795,Z 456.052,A -85,B 0,C 180,E1 -27254.533,E2 -27254.533} C_VEL
LIN {X 0,Y 96.952,Z 456.017,A -85,B 0,C 180,E1 -27255.549,E2 -27255.549} C_VEL
LIN {X 0,Y 98.377,Z 457.158,A -85,B 0,C 180,E1 -27256.566,E2 -27256.566} C_VEL
LIN {X 0,Y 99,Z 461.4,A -85,B 0,C 180,E1 -27258.264,E2 -27258.264} C_VEL
LIN {X 0,Y 99.306,Z 471.237,A -85,B 0,C 180,E1 -27262.21,E2 -27262.21} C_VEL
LIN {X 0,Y 98.924,Z 479.545,A -85,B 0,C 180,E1 -27265.917,E2 -27265.917} C_VEL
LIN {X 0,Y 98.498,Z 482.514,A -85,B 0,C 180,E1 -27267.31,E2 -27267.31} C_VEL
LIN {X 0,Y 95.248,Z 490.517,A -85,B 0,C 180,E1 -27271.048,E2 -27271.048} C_VEL
LIN {X 0,Y 91.839,Z 498.43,A -85,B 0,C 180,E1 -27275.845,E2 -27275.845} C_VEL
LIN {X 0,Y 88.837,Z 505.418,A -85,B 0,C 180,E1 -27281.396,E2 -27281.396} C_VEL
LIN {X 0,Y 86.627,Z 510.686,A -85,B 0,C 180,E1 -27286.815,E2 -27286.815} C_VEL
LIN {X 0,Y 84.701,Z 516.281,A -85,B 0,C 180,E1 -27294.499,E2 -27294.499} C_VEL
LIN {X 0,Y 83.972,Z 520.722,A -85,B 0,C 180,E1 -27303.184,E2 -27303.184} C_VEL
LIN {X 0,Y 85.026,Z 523.575,A -85,B 0,C 180,E1 -27311.936,E2 -27311.936} C_VEL
LIN {X 0,Y 87.7,Z 524.889,A -85,B 0,C 180,E1 -27320.128,E2 -27320.128} C_VEL
LIN {X 0,Y 91.876,Z 524.828,A -85,B 0,C 180,E1 -27327.626,E2 -27327.626} C_VEL
LIN {X 0,Y 97.192,Z 523.488,A -85,B 0,C 180,E1 -27334.289,E2 -27334.289} C_VEL
LIN {X 0,Y 104.243,Z 520.504,A -85,B 0,C 180,E1 -27340.682,E2 -27340.682} C_VEL
LIN {X 0,Y 111.05,Z 516.728,A -85,B 0,C 180,E1 -27345.337,E2 -27345.337} C_VEL
LIN {X 0,Y 119.436,Z 510.91,A -85,B 0,C 180,E1 -27349.833,E2 -27349.833} C_VEL
LIN {X 0,Y 121.081,Z 509.636,A -85,B 0,C 180,E1 -27350.607,E2 -27350.607} C_VEL
LIN {X 0,Y 123.166,Z 507.646,A -85,B 0,C 180,E1 -27352.11,E2 -27352.11} C_VEL
LIN {X 0,Y 124.323,Z 506.149,A -85,B 0,C 180,E1 -27353.509,E2 -27353.509} C_VEL
LIN {X 0,Y 125.158,Z 504.74,A -85,B 0,C 180,E1 -27355.169,E2 -27355.169} C_VEL
LIN {X 0,Y 126.403,Z 501.448,A -85,B 0,C 180,E1 -27360.001,E2 -27360.001} C_VEL
LIN {X 0,Y 126.97,Z 499.764,A -85,B 0,C 180,E1 -27363.174,E2 -27363.174} C_VEL
LIN {X 0,Y 127.236,Z 498.526,A -85,B 0,C 180,E1 -27366.344,E2 -27366.344} C_VEL
LIN {X 0,Y 127.274,Z 497.751,A -85,B 0,C 180,E1 -27372.762,E2 -27372.762} C_VEL
LIN {X 0,Y 127.165,Z 498.136,A -85,B 0,C 180,E1 -27376.043,E2 -27376.043} C_VEL
LIN {X 0,Y 126.934,Z 499.156,A -85,B 0,C 180,E1 -27379.763,E2 -27379.763} C_VEL
LIN {X 0,Y 126.862,Z 500.337,A -85,B 0,C 180,E1 -27382.818,E2 -27382.818} C_VEL
LIN {X 0,Y 126.641,Z 502.822,A -85,B 0,C 180,E1 -27387.404,E2 -27387.404} C_VEL
LIN {X 0,Y 126.057,Z 505.959,A -85,B 0,C 180,E1 -27391.609,E2 -27391.609} C_VEL
LIN {X 0,Y 125.245,Z 509.09,A -85,B 0,C 180,E1 -27395.246,E2 -27395.246} C_VEL
LIN {X 0,Y 121.814,Z 512.913,A -85,B 0,C 180,E1 -27397.519,E2 -27397.519} C_VEL
LIN {X 0,Y 115.568,Z 518.152,A -85,B 0,C 180,E1 -27400.535,E2 -27400.535} C_VEL
LIN {X 0,Y 108.317,Z 523.277,A -85,B 0,C 180,E1 -27404.475,E2 -27404.475} C_VEL
LIN {X 0,Y 100.266,Z 528.122,A -85,B 0,C 180,E1 -27410.449,E2 -27410.449} C_VEL
LIN {X 0,Y 96.322,Z 530.165,A -85,B 0,C 180,E1 -27414.301,E2 -27414.301} C_VEL
LIN {X 0,Y 90.192,Z 532.603,A -85,B 0,C 180,E1 -27422.137,E2 -27422.137} C_VEL
LIN {X 0,Y 87.821,Z 533.233,A -85,B 0,C 180,E1 -27426.425,E2 -27426.425} C_VEL
LIN {X 0,Y 84.964,Z 533.275,A -85,B 0,C 180,E1 -27435.643,E2 -27435.643} C_VEL
LIN {X 0,Y 84.375,Z 532.732,A -85,B 0,C 180,E1 -27440.421,E2 -27440.421} C_VEL
LIN {X 0,Y 84.788,Z 530.8,A -85,B 0,C 180,E1 -27448.808,E2 -27448.808} C_VEL
LIN {X 0,Y 84.696,Z 534.567,A -85,B 0,C 180,E1 -27454.77,E2 -27454.77} C_VEL
LIN {X 0,Y 85.443,Z 539.064,A -85,B 0,C 180,E1 -27464.296,E2 -27464.296} C_VEL
LIN {X 0,Y 88.407,Z 542.056,A -85,B 0,C 180,E1 -27473.431,E2 -27473.431} C_VEL
LIN {X 0,Y 93.656,Z 543.758,A -85,B 0,C 180,E1 -27481.698,E2 -27481.698} C_VEL
LIN {X 0,Y 100.893,Z 544.196,A -85,B 0,C 180,E1 -27488.833,E2 -27488.833} C_VEL
LIN {X 0,Y 109.571,Z 543.326,A -85,B 0,C 180,E1 -27494.884,E2 -27494.884} C_VEL
LIN {X 0,Y 119.413,Z 541.188,A -85,B 0,C 180,E1 -27499.927,E2 -27499.927} C_VEL
LIN {X 0,Y 124.697,Z 539.644,A -85,B 0,C 180,E1 -27502.106,E2 -27502.106} C_VEL
LIN {X 0,Y 136.022,Z 535.478,A -85,B 0,C 180,E1 -27505.77,E2 -27505.77} C_VEL
LIN {X 0,Y 143.876,Z 531.853,A -85,B 0,C 180,E1 -27507.864,E2 -27507.864} C_VEL
LIN {X 0,Y 144.268,Z 531.478,A -85,B 0,C 180,E1 -27509.399,E2 -27509.399} C_VEL
LIN {X 0,Y 144.008,Z 531.405,A -85,B 0,C 180,E1 -27511.466,E2 -27511.466} C_VEL
LIN {X 0,Y 143.487,Z 531.593,A -85,B 0,C 180,E1 -27513.843,E2 -27513.843} C_VEL
LIN {X 0,Y 142.3,Z 532.17,A -85,B 0,C 180,E1 -27515.177,E2 -27515.177} C_VEL
LIN {X 0,Y 132.186,Z 536.219,A -85,B 0,C 180,E1 -27518.149,E2 -27518.149} C_VEL
LIN {X 0,Y 125.764,Z 538.26,A -85,B 0,C 180,E1 -27520.408,E2 -27520.408} C_VEL
LIN {X 0,Y 116.867,Z 540.407,A -85,B 0,C 180,E1 -27524.216,E2 -27524.216} C_VEL
LIN {X 0,Y 107.18,Z 541.684,A -85,B 0,C 180,E1 -27529.642,E2 -27529.642} C_VEL
LIN {X 0,Y 98.611,Z 541.61,A -85,B 0,C 180,E1 -27536.297,E2 -27536.297} C_VEL
LIN {X 0,Y 91.55,Z 539.988,A -85,B 0,C 180,E1 -27544.401,E2 -27544.401} C_VEL
LIN {X 0,Y 86.721,Z 536.908,A -85,B 0,C 180,E1 -27553.43,E2 -27553.43} C_VEL
LIN {X 0,Y 84.141,Z 532.169,A -85,B 0,C 180,E1 -27563.227,E2 -27563.227} C_VEL
LIN {X 0,Y 83.684,Z 527.779,A -85,B 0,C 180,E1 -27570.256,E2 -27570.256} C_VEL
LIN {X 0,Y 84.209,Z 522.366,A -85,B 0,C 180,E1 -27577.232,E2 -27577.232} C_VEL
LIN {X 0,Y 84.797,Z 518.587,A -85,B 0,C 180,E1 -27581.302,E2 -27581.302} C_VEL
LIN {X 0,Y 84.892,Z 516.335,A -85,B 0,C 180,E1 -27583.481,E2 -27583.481} C_VEL
LIN {X 0,Y 83.978,Z 511.467,A -85,B 0,C 180,E1 -27587.678,E2 -27587.678} C_VEL
LIN {X 0,Y 82.26,Z 502.071,A -85,B 0,C 180,E1 -27594.721,E2 -27594.721} C_VEL
LIN {X 0,Y 82.9,Z 497.706,A -85,B 0,C 180,E1 -27597.497,E2 -27597.497} C_VEL
LIN {X 0,Y 86.46,Z 486.309,A -85,B 0,C 180,E1 -27603.396,E2 -27603.396} C_VEL
LIN {X 0,Y 87.988,Z 480.562,A -85,B 0,C 180,E1 -27605.816,E2 -27605.816} C_VEL
LIN {X 0,Y 87.573,Z 468.422,A -85,B 0,C 180,E1 -27610.657,E2 -27610.657} C_VEL
LIN {X 0,Y 87.205,Z 462.246,A -85,B 0,C 180,E1 -27612.906,E2 -27612.906} C_VEL
LIN {X 0,Y 87.892,Z 463.072,A -85,B 0,C 180,E1 -27613.64,E2 -27613.64} C_VEL
LIN {X 0,Y 93.001,Z 464.68,A -85,B 0,C 180,E1 -27616.887,E2 -27616.887} C_VEL
LIN {X 0,Y 92.986,Z 473.379,A -85,B 0,C 180,E1 -27620.749,E2 -27620.749} C_VEL
LIN {X 0,Y 92.342,Z 481.655,A -85,B 0,C 180,E1 -27624.804,E2 -27624.804} C_VEL
LIN {X 0,Y 91.102,Z 485.381,A -85,B 0,C 180,E1 -27626.562,E2 -27626.562} C_VEL
LIN {X 0,Y 87.346,Z 493.865,A -85,B 0,C 180,E1 -27631.142,E2 -27631.142} C_VEL
LIN {X 0,Y 83.448,Z 502.284,A -85,B 0,C 180,E1 -27637.257,E2 -27637.257} C_VEL
LIN {X 0,Y 80.462,Z 508.795,A -85,B 0,C 180,E1 -27643.617,E2 -27643.617} C_VEL
LIN {X 0,Y 78.219,Z 514.444,A -85,B 0,C 180,E1 -27651.051,E2 -27651.051} C_VEL
LIN {X 0,Y 76.955,Z 519.444,A -85,B 0,C 180,E1 -27660.138,E2 -27660.138} C_VEL
LIN {X 0,Y 77.42,Z 522.866,A -85,B 0,C 180,E1 -27669.437,E2 -27669.437} C_VEL
LIN {X 0,Y 78.746,Z 524.354,A -85,B 0,C 180,E1 -27675.543,E2 -27675.543} C_VEL
LIN {X 0,Y 81.589,Z 525.336,A -85,B 0,C 180,E1 -27682.919,E2 -27682.919} C_VEL
LIN {X 0,Y 86.323,Z 525.248,A -85,B 0,C 180,E1 -27690.761,E2 -27690.761} C_VEL
LIN {X 0,Y 92.253,Z 523.869,A -85,B 0,C 180,E1 -27697.612,E2 -27697.612} C_VEL
LIN {X 0,Y 99.318,Z 521.153,A -85,B 0,C 180,E1 -27703.559,E2 -27703.559} C_VEL
LIN {X 0,Y 107.477,Z 516.976,A -85,B 0,C 180,E1 -27708.722,E2 -27708.722} C_VEL
LIN {X 0,Y 116.336,Z 511.176,A -85,B 0,C 180,E1 -27713.062,E2 -27713.062} C_VEL
LIN {X 0,Y 117.72,Z 510.009,A -85,B 0,C 180,E1 -27714.004,E2 -27714.004} C_VEL
LIN {X 0,Y 118.568,Z 509.121,A -85,B 0,C 180,E1 -27714.9,E2 -27714.9} C_VEL
LIN {X 0,Y 119.62,Z 507.602,A -85,B 0,C 180,E1 -27717.012,E2 -27717.012} C_VEL
LIN {X 0,Y 120.553,Z 505.87,A -85,B 0,C 180,E1 -27720.001,E2 -27720.001} C_VEL
LIN {X 0,Y 121.324,Z 504.245,A -85,B 0,C 180,E1 -27723.322,E2 -27723.322} C_VEL
LIN {X 0,Y 121.82,Z 503.107,A -85,B 0,C 180,E1 -27726.627,E2 -27726.627} C_VEL
LIN {X 0,Y 121.855,Z 502.563,A -85,B 0,C 180,E1 -27731.385,E2 -27731.385} C_VEL
LIN {X 0,Y 121.894,Z 502.525,A -85,B 0,C 180,E1 -27733.335,E2 -27733.335} C_VEL
LIN {X 0,Y 121.723,Z 503.055,A -85,B 0,C 180,E1 -27736.781,E2 -27736.781} C_VEL
LIN {X 0,Y 121.425,Z 504.7,A -85,B 0,C 180,E1 -27742.193,E2 -27742.193} C_VEL
LIN {X 0,Y 121.165,Z 506.342,A -85,B 0,C 180,E1 -27745.788,E2 -27745.788} C_VEL
LIN {X 0,Y 120.551,Z 508.38,A -85,B 0,C 180,E1 -27749.034,E2 -27749.034} C_VEL
LIN {X 0,Y 119.644,Z 511.266,A -85,B 0,C 180,E1 -27753.037,E2 -27753.037} C_VEL
LIN {X 0,Y 118.737,Z 512.462,A -85,B 0,C 180,E1 -27754.055,E2 -27754.055} C_VEL
LIN {X 0,Y 115.092,Z 515.658,A -85,B 0,C 180,E1 -27756.007,E2 -27756.007} C_VEL
LIN {X 0,Y 105.929,Z 521.985,A -85,B 0,C 180,E1 -27760.287,E2 -27760.287} C_VEL
LIN {X 0,Y 98.817,Z 526.151,A -85,B 0,C 180,E1 -27764.681,E2 -27764.681} C_VEL
LIN {X 0,Y 94.366,Z 528.415,A -85,B 0,C 180,E1 -27768.14,E2 -27768.14} C_VEL
LIN {X 0,Y 87.041,Z 531.407,A -85,B 0,C 180,E1 -27775.597,E2 -27775.597} C_VEL
LIN {X 0,Y 83.959,Z 532.346,A -85,B 0,C 180,E1 -27779.865,E2 -27779.865} C_VEL
LIN {X 0,Y 81.334,Z 532.853,A -85,B 0,C 180,E1 -27784.415,E2 -27784.415} C_VEL
LIN {X 0,Y 78.081,Z 532.758,A -85,B 0,C 180,E1 -27794.346,E2 -27794.346} C_VEL
LIN {X 0,Y 77.334,Z 531.037,A -85,B 0,C 180,E1 -27804.798,E2 -27804.798} C_VEL
LIN {X 0,Y 77.85,Z 529.802,A -85,B 0,C 180,E1 -27809.582,E2 -27809.582} C_VEL
LIN {X 0,Y 77.743,Z 533.629,A -85,B 0,C 180,E1 -27816.047,E2 -27816.047} C_VEL
LIN {X 0,Y 78.644,Z 537.95,A -85,B 0,C 180,E1 -27825.562,E2 -27825.562} C_VEL
LIN {X 0,Y 81.955,Z 541.257,A -85,B 0,C 180,E1 -27835.401,E2 -27835.401} C_VEL
LIN {X 0,Y 87.703,Z 543.225,A -85,B 0,C 180,E1 -27844.132,E2 -27844.132} C_VEL
LIN {X 0,Y 95.471,Z 543.937,A -85,B 0,C 180,E1 -27851.504,E2 -27851.504} C_VEL
LIN {X 0,Y 104.66,Z 543.404,A -85,B 0,C 180,E1 -27857.628,E2 -27857.628} C_VEL
LIN {X 0,Y 114.986,Z 541.636,A -85,B 0,C 180,E1 -27862.625,E2 -27862.625} C_VEL
LIN {X 0,Y 120.484,Z 540.269,A -85,B 0,C 180,E1 -27864.761,E2 -27864.761} C_VEL
LIN {X 0,Y 132.2,Z 536.476,A -85,B 0,C 180,E1 -27868.287,E2 -27868.287} C_VEL
LIN {X 0,Y 135.243,Z 535.324,A -85,B 0,C 180,E1 -27869.04,E2 -27869.04} C_VEL
LIN {X 0,Y 137.639,Z 534.257,A -85,B 0,C 180,E1 -27870.242,E2 -27870.242} C_VEL
LIN {X 0,Y 137.188,Z 534.287,A -85,B 0,C 180,E1 -27872.543,E2 -27872.543} C_VEL
LIN {X 0,Y 132.532,Z 535.993,A -85,B 0,C 180,E1 -27874.367,E2 -27874.367} C_VEL
LIN {X 0,Y 121.41,Z 539.283,A -85,B 0,C 180,E1 -27877.863,E2 -27877.863} C_VEL
LIN {X 0,Y 110.688,Z 541.318,A -85,B 0,C 180,E1 -27882.274,E2 -27882.274} C_VEL
LIN {X 0,Y 100.595,Z 542.062,A -85,B 0,C 180,E1 -27887.9,E2 -27887.9} C_VEL
LIN {X 0,Y 91.747,Z 541.452,A -85,B 0,C 180,E1 -27894.853,E2 -27894.853} C_VEL
LIN {X 0,Y 84.499,Z 539.337,A -85,B 0,C 180,E1 -27903.406,E2 -27903.406} C_VEL
LIN {X 0,Y 79.471,Z 535.677,A -85,B 0,C 180,E1 -27913.354,E2 -27913.354} C_VEL
LIN {X 0,Y 77.361,Z 531.863,A -85,B 0,C 180,E1 -27921.307,E2 -27921.307} C_VEL
LIN {X 0,Y 76.677,Z 526.552,A -85,B 0,C 180,E1 -27930.271,E2 -27930.271} C_VEL
LIN {X 0,Y 77.288,Z 520.712,A -85,B 0,C 180,E1 -27938.085,E2 -27938.085} C_VEL
LIN {X 0,Y 78.631,Z 513.513,A -85,B 0,C 180,E1 -27945.643,E2 -27945.643} C_VEL
LIN {X 0,Y 81.06,Z 503.959,A -85,B 0,C 180,E1 -27953.414,E2 -27953.414} C_VEL
LIN {X 0,Y 82.9,Z 497.706,A -85,B 0,C 180,E1 -27957.497,E2 -27957.497} C_VEL
LIN {X 0,Y 83.592,Z 493.273,A -85,B 0,C 180,E1 -27960.074,E2 -27960.074} C_VEL
LIN {X 0,Y 83.323,Z 488.675,A -85,B 0,C 180,E1 -27962.637,E2 -27962.637} C_VEL
LIN {X 0,Y 81.579,Z 479.048,A -85,B 0,C 180,E1 -27967.653,E2 -27967.653} C_VEL
LIN {X 0,Y 80.87,Z 472.171,A -85,B 0,C 180,E1 -27970.814,E2 -27970.814} C_VEL
LIN {X 0,Y 80.805,Z 468.729,A -85,B 0,C 180,E1 -27972.323,E2 -27972.323} C_VEL
LIN {X 0,Y 81.003,Z 469.067,A -85,B 0,C 180,E1 -27972.623,E2 -27972.623} C_VEL
LIN {X 0,Y 86.839,Z 469.84,A -85,B 0,C 180,E1 -27976.203,E2 -27976.203} C_VEL
LIN {X 0,Y 86.752,Z 474.982,A -85,B 0,C 180,E1 -27978.839,E2 -27978.839} C_VEL
LIN {X 0,Y 85.954,Z 482.531,A -85,B 0,C 180,E1 -27982.875,E2 -27982.875} C_VEL
LIN {X 0,Y 84.133,Z 487.149,A -85,B 0,C 180,E1 -27985.198,E2 -27985.198} C_VEL
LIN {X 0,Y 80.239,Z 495.224,A -85,B 0,C 180,E1 -27989.989,E2 -27989.989} C_VEL
LIN {X 0,Y 76.221,Z 503.446,A -85,B 0,C 180,E1 -27996.606,E2 -27996.606} C_VEL
LIN {X 0,Y 72.703,Z 510.757,A -85,B 0,C 180,E1 -28004.842,E2 -28004.842} C_VEL
LIN {X 0,Y 70.608,Z 516.255,A -85,B 0,C 180,E1 -28013.448,E2 -28013.448} C_VEL
LIN {X 0,Y 69.791,Z 520.735,A -85,B 0,C 180,E1 -28023.349,E2 -28023.349} C_VEL
LIN {X 0,Y 71.076,Z 523.911,A -85,B 0,C 180,E1 -28033.782,E2 -28033.782} C_VEL
LIN {X 0,Y 73.04,Z 525.182,A -85,B 0,C 180,E1 -28040.312,E2 -28040.312} C_VEL
LIN {X 0,Y 75.843,Z 525.804,A -85,B 0,C 180,E1 -28046.487,E2 -28046.487} C_VEL
LIN {X 0,Y 81.063,Z 525.669,A -85,B 0,C 180,E1 -28054.312,E2 -28054.312} C_VEL
LIN {X 0,Y 88.598,Z 523.982,A -85,B 0,C 180,E1 -28062.119,E2 -28062.119} C_VEL
LIN {X 0,Y 95.448,Z 521.519,A -85,B 0,C 180,E1 -28067.24,E2 -28067.24} C_VEL
LIN {X 0,Y 102.012,Z 518.452,A -85,B 0,C 180,E1 -28071.151,E2 -28071.151} C_VEL
LIN {X 0,Y 109.383,Z 514.242,A -85,B 0,C 180,E1 -28074.7,E2 -28074.7} C_VEL
LIN {X 0,Y 111.856,Z 512.641,A -85,B 0,C 180,E1 -28075.751,E2 -28075.751} C_VEL
LIN {X 0,Y 112.752,Z 511.932,A -85,B 0,C 180,E1 -28076.428,E2 -28076.428} C_VEL
LIN {X 0,Y 114.382,Z 509.934,A -85,B 0,C 180,E1 -28080.001,E2 -28080.001} C_VEL
LIN {X 0,Y 115.443,Z 508.407,A -85,B 0,C 180,E1 -28083.491,E2 -28083.491} C_VEL
LIN {X 0,Y 116.139,Z 507.326,A -85,B 0,C 180,E1 -28086.953,E2 -28086.953} C_VEL
LIN {X 0,Y 116.232,Z 506.997,A -85,B 0,C 180,E1 -28090.452,E2 -28090.452} C_VEL
LIN {X 0,Y 116.19,Z 507.129,A -85,B 0,C 180,E1 -28094.618,E2 -28094.618} C_VEL
LIN {X 0,Y 116.003,Z 507.678,A -85,B 0,C 180,E1 -28097.635,E2 -28097.635} C_VEL
LIN {X 0,Y 115.727,Z 508.699,A -85,B 0,C 180,E1 -28101.37,E2 -28101.37} C_VEL
LIN {X 0,Y 115.316,Z 510.27,A -85,B 0,C 180,E1 -28105.254,E2 -28105.254} C_VEL
LIN {X 0,Y 114.054,Z 513.262,A -85,B 0,C 180,E1 -28110.399,E2 -28110.399} C_VEL
LIN {X 0,Y 112.397,Z 515.217,A -85,B 0,C 180,E1 -28112.438,E2 -28112.438} C_VEL
LIN {X 0,Y 104.163,Z 520.728,A -85,B 0,C 180,E1 -28115.954,E2 -28115.954} C_VEL
LIN {X 0,Y 96.388,Z 525.059,A -85,B 0,C 180,E1 -28120.056,E2 -28120.056} C_VEL
LIN {X 0,Y 88.656,Z 528.623,A -85,B 0,C 180,E1 -28125.519,E2 -28125.519} C_VEL
LIN {X 0,Y 81.26,Z 531.231,A -85,B 0,C 180,E1 -28132.756,E2 -28132.756} C_VEL
LIN {X 0,Y 74.97,Z 532.475,A -85,B 0,C 180,E1 -28142.063,E2 -28142.063} C_VEL
LIN {X 0,Y 72.788,Z 532.542,A -85,B 0,C 180,E1 -28147.295,E2 -28147.295} C_VEL
LIN {X 0,Y 70.401,Z 531.443,A -85,B 0,C 180,E1 -28158.496,E2 -28158.496} C_VEL
LIN {X 0,Y 70.419,Z 529.773,A -85,B 0,C 180,E1 -28166.425,E2 -28166.425} C_VEL
LIN {X 0,Y 70.924,Z 528.739,A -85,B 0,C 180,E1 -28170.488,E2 -28170.488} C_VEL
LIN {X 0,Y 70.851,Z 532.5,A -85,B 0,C 180,E1 -28177.265,E2 -28177.265} C_VEL
LIN {X 0,Y 71.905,Z 536.761,A -85,B 0,C 180,E1 -28187.063,E2 -28187.063} C_VEL
LIN {X 0,Y 75.649,Z 540.33,A -85,B 0,C 180,E1 -28197.691,E2 -28197.691} C_VEL
LIN {X 0,Y 81.947,Z 542.595,A -85,B 0,C 180,E1 -28206.907,E2 -28206.907} C_VEL
LIN {X 0,Y 90.282,Z 543.64,A -85,B 0,C 180,E1 -28214.488,E2 -28214.488} C_VEL
LIN {X 0,Y 100.011,Z 543.434,A -85,B 0,C 180,E1 -28220.636,E2 -28220.636} C_VEL
LIN {X 0,Y 110.825,Z 541.97,A -85,B 0,C 180,E1 -28225.54,E2 -28225.54} C_VEL
LIN {X 0,Y 116.553,Z 540.784,A -85,B 0,C 180,E1 -28227.597,E2 -28227.597} C_VEL
LIN {X 0,Y 128.647,Z 537.403,A -85,B 0,C 180,E1 -28230.948,E2 -28230.948} C_VEL
LIN {X 0,Y 127.099,Z 537.792,A -85,B 0,C 180,E1 -28232.226,E2 -28232.226} C_VEL
LIN {X 0,Y 115.703,Z 540.526,A -85,B 0,C 180,E1 -28235.677,E2 -28235.677} C_VEL
LIN {X 0,Y 104.222,Z 542.058,A -85,B 0,C 180,E1 -28240.294,E2 -28240.294} C_VEL
LIN {X 0,Y 94.252,Z 542.242,A -85,B 0,C 180,E1 -28245.812,E2 -28245.812} C_VEL
LIN {X 0,Y 84.957,Z 541.097,A -85,B 0,C 180,E1 -28253.146,E2 -28253.146} C_VEL
LIN {X 0,Y 77.385,Z 538.465,A -85,B 0,C 180,E1 -28262.323,E2 -28262.323} C_VEL
LIN {X 0,Y 72.225,Z 534.209,A -85,B 0,C 180,E1 -28273.278,E2 -28273.278} C_VEL
LIN {X 0,Y 70.016,Z 529.12,A -85,B 0,C 180,E1 -28283.67,E2 -28283.67} C_VEL
LIN {X 0,Y 69.845,Z 523.034,A -85,B 0,C 180,E1 -28293.481,E2 -28293.481} C_VEL
LIN {X 0,Y 70.559,Z 517.8,A -85,B 0,C 180,E1 -28300.345,E2 -28300.345} C_VEL
LIN {X 0,Y 72.188,Z 510.205,A -85,B 0,C 180,E1 -28308.365,E2 -28308.365} C_VEL
LIN {X 0,Y 74.859,Z 500.642,A -85,B 0,C 180,E1 -28316.107,E2 -28316.107} C_VEL
LIN {X 0,Y 78.222,Z 490.194,A -85,B 0,C 180,E1 -28322.524,E2 -28322.524} C_VEL
LIN {X 0,Y 80.677,Z 482.591,A -85,B 0,C 180,E1 -28326.15,E2 -28326.15} C_VEL
LIN {X 0,Y 81.025,Z 479.221,A -85,B 0,C 180,E1 -28327.687,E2 -28327.687} C_VEL
LIN {X 0,Y 80.87,Z 472.171,A -85,B 0,C 180,E1 -28330.814,E2 -28330.814} C_VEL
LIN {X 0,Y 80.806,Z 471.586,A -85,B 0,C 180,E1 -28331.711,E2 -28331.711} C_VEL
LIN {X 0,Y 80.679,Z 472.406,A -85,B 0,C 180,E1 -28333.526,E2 -28333.526} C_VEL
LIN {X 0,Y 80.46,Z 476.248,A -85,B 0,C 180,E1 -28336.44,E2 -28336.44} C_VEL
LIN {X 0,Y 79.702,Z 482.576,A -85,B 0,C 180,E1 -28340.12,E2 -28340.12} C_VEL
LIN {X 0,Y 78.428,Z 486.271,A -85,B 0,C 180,E1 -28342.178,E2 -28342.178} C_VEL
LIN {X 0,Y 74.161,Z 494.677,A -85,B 0,C 180,E1 -28347.272,E2 -28347.272} C_VEL
LIN {X 0,Y 69.777,Z 503,A -85,B 0,C 180,E1 -28354.275,E2 -28354.275} C_VEL
LIN {X 0,Y 66.24,Z 509.808,A -85,B 0,C 180,E1 -28362.237,E2 -28362.237} C_VEL
LIN {X 0,Y 64.245,Z 514.257,A -85,B 0,C 180,E1 -28369.143,E2 -28369.143} C_VEL
LIN {X 0,Y 62.762,Z 519.495,A -85,B 0,C 180,E1 -28380.237,E2 -28380.237} C_VEL
LIN {X 0,Y 63.45,Z 523.215,A -85,B 0,C 180,E1 -28391.631,E2 -28391.631} C_VEL
LIN {X 0,Y 65.499,Z 525.058,A -85,B 0,C 180,E1 -28399.927,E2 -28399.927} C_VEL
LIN {X 0,Y 69.99,Z 526.228,A -85,B 0,C 180,E1 -28409.865,E2 -28409.865} C_VEL
LIN {X 0,Y 76.13,Z 526.102,A -85,B 0,C 180,E1 -28418.332,E2 -28418.332} C_VEL
LIN {X 0,Y 83.468,Z 524.675,A -85,B 0,C 180,E1 -28425.37,E2 -28425.37} C_VEL
LIN {X 0,Y 92.374,Z 521.746,A -85,B 0,C 180,E1 -28431.445,E2 -28431.445} C_VEL
LIN {X 0,Y 101.343,Z 517.664,A -85,B 0,C 180,E1 -28436.025,E2 -28436.025} C_VEL
LIN {X 0,Y 105.48,Z 515.395,A -85,B 0,C 180,E1 -28437.798,E2 -28437.798} C_VEL
LIN {X 0,Y 107.86,Z 513.726,A -85,B 0,C 180,E1 -28440.001,E2 -28440.001} C_VEL
LIN {X 0,Y 109.283,Z 512.233,A -85,B 0,C 180,E1 -28443.689,E2 -28443.689} C_VEL
LIN {X 0,Y 110.218,Z 511.225,A -85,B 0,C 180,E1 -28447.328,E2 -28447.328} C_VEL
LIN {X 0,Y 110.328,Z 510.991,A -85,B 0,C 180,E1 -28451.018,E2 -28451.018} C_VEL
LIN {X 0,Y 110.297,Z 511.18,A -85,B 0,C 180,E1 -28454.767,E2 -28454.767} C_VEL
LIN {X 0,Y 109.959,Z 511.925,A -85,B 0,C 180,E1 -28458.638,E2 -28458.638} C_VEL
LIN {X 0,Y 109.55,Z 513.09,A -85,B 0,C 180,E1 -28462.64,E2 -28462.64} C_VEL
LIN {X 0,Y 108.642,Z 514.971,A -85,B 0,C 180,E1 -28466.927,E2 -28466.927} C_VEL
LIN {X 0,Y 107.824,Z 516.239,A -85,B 0,C 180,E1 -28469.218,E2 -28469.218} C_VEL
LIN {X 0,Y 105.918,Z 517.674,A -85,B 0,C 180,E1 -28470.41,E2 -28470.41} C_VEL
LIN {X 0,Y 97.375,Z 522.59,A -85,B 0,C 180,E1 -28473.919,E2 -28473.919} C_VEL
LIN {X 0,Y 89.381,Z 526.381,A -85,B 0,C 180,E1 -28478.178,E2 -28478.178} C_VEL
LIN {X 0,Y 83.045,Z 528.859,A -85,B 0,C 180,E1 -28482.614,E2 -28482.614} C_VEL
LIN {X 0,Y 75.712,Z 531.003,A -85,B 0,C 180,E1 -28489.492,E2 -28489.492} C_VEL
LIN {X 0,Y 68.761,Z 532.094,A -85,B 0,C 180,E1 -28499.282,E2 -28499.282} C_VEL
LIN {X 0,Y 64.501,Z 531.589,A -85,B 0,C 180,E1 -28510.936,E2 -28510.936} C_VEL
LIN {X 0,Y 63.447,Z 530.772,A -85,B 0,C 180,E1 -28517.215,E2 -28517.215} C_VEL
LIN {X 0,Y 63.384,Z 528.895,A -85,B 0,C 180,E1 -28526.335,E2 -28526.335} C_VEL
LIN {X 0,Y 64.027,Z 527.579,A -85,B 0,C 180,E1 -28531.593,E2 -28531.593} C_VEL
LIN {X 0,Y 64.004,Z 531.249,A -85,B 0,C 180,E1 -28538.776,E2 -28538.776} C_VEL
LIN {X 0,Y 65.252,Z 535.462,A -85,B 0,C 180,E1 -28548.865,E2 -28548.865} C_VEL
LIN {X 0,Y 69.485,Z 539.326,A -85,B 0,C 180,E1 -28560.393,E2 -28560.393} C_VEL
LIN {X 0,Y 76.412,Z 541.913,A -85,B 0,C 180,E1 -28570.092,E2 -28570.092} C_VEL
LIN {X 0,Y 85.368,Z 543.224,A -85,B 0,C 180,E1 -28577.825,E2 -28577.825} C_VEL
LIN {X 0,Y 96.886,Z 543.276,A -85,B 0,C 180,E1 -28584.526,E2 -28584.526} C_VEL
LIN {X 0,Y 106.983,Z 542.244,A -85,B 0,C 180,E1 -28588.663,E2 -28588.663} C_VEL
LIN {X 0,Y 112.916,Z 541.243,A -85,B 0,C 180,E1 -28590.633,E2 -28590.633} C_VEL
LIN {X 0,Y 114.472,Z 540.902,A -85,B 0,C 180,E1 -28591.889,E2 -28591.889} C_VEL
LIN {X 0,Y 103.035,Z 542.306,A -85,B 0,C 180,E1 -28595.84,E2 -28595.84} C_VEL
LIN {X 0,Y 96.631,Z 542.558,A -85,B 0,C 180,E1 -28598.674,E2 -28598.674} C_VEL
LIN {X 0,Y 87.983,Z 542.223,A -85,B 0,C 180,E1 -28603.475,E2 -28603.475} C_VEL
LIN {X 0,Y 78.244,Z 540.527,A -85,B 0,C 180,E1 -28611.192,E2 -28611.192} C_VEL
LIN {X 0,Y 70.307,Z 537.376,A -85,B 0,C 180,E1 -28621.094,E2 -28621.094} C_VEL
LIN {X 0,Y 65.221,Z 532.825,A -85,B 0,C 180,E1 -28632.443,E2 -28632.443} C_VEL
LIN {X 0,Y 63.085,Z 527.849,A -85,B 0,C 180,E1 -28642.889,E2 -28642.889} C_VEL
LIN {X 0,Y 62.911,Z 521.381,A -85,B 0,C 180,E1 -28653.954,E2 -28653.954} C_VEL
LIN {X 0,Y 64.005,Z 514.359,A -85,B 0,C 180,E1 -28663.333,E2 -28663.333} C_VEL
LIN {X 0,Y 65.746,Z 507.051,A -85,B 0,C 180,E1 -28671.055,E2 -28671.055} C_VEL
LIN {X 0,Y 68.637,Z 497.704,A -85,B 0,C 180,E1 -28678.742,E2 -28678.742} C_VEL
LIN {X 0,Y 72.332,Z 486.893,A -85,B 0,C 180,E1 -28685.424,E2 -28685.424} C_VEL
LIN {X 0,Y 74.142,Z 480.885,A -85,B 0,C 180,E1 -28688.394,E2 -28688.394} C_VEL
LIN {X 0,Y 74.101,Z 474.617,A -85,B 0,C 180,E1 -28691.515,E2 -28691.515} C_VEL
LIN {X 0,Y 76.662,Z 475.873,A -85,B 0,C 180,E1 -28694.025,E2 -28694.025} C_VEL
LIN {X 0,Y 79.854,Z 475.248,A -85,B 0,C 180,E1 -28695.486,E2 -28695.486} C_VEL
LIN {X 0,Y 80.578,Z 476.519,A -85,B 0,C 180,E1 -28696.67,E2 -28696.67} C_VEL
LIN {X 0,Y 79.6,Z 483.628,A -85,B 0,C 180,E1 -28700.811,E2 -28700.811} C_VEL
LIN {X 0,Y 78.428,Z 486.271,A -85,B 0,C 180,E1 -28702.178,E2 -28702.178} C_VEL
LIN {X 0,Y 75.722,Z 490.625,A -85,B 0,C 180,E1 -28704.373,E2 -28704.373} C_VEL
LIN {X 0,Y 69.742,Z 497.163,A -85,B 0,C 180,E1 -28707.879,E2 -28707.879} C_VEL
LIN {X 0,Y 63.731,Z 503.16,A -85,B 0,C 180,E1 -28712.383,E2 -28712.383} C_VEL
LIN {X 0,Y 61.128,Z 506.58,A -85,B 0,C 180,E1 -28716.12,E2 -28716.12} C_VEL
LIN {X 0,Y 58.108,Z 512.349,A -85,B 0,C 180,E1 -28724.641,E2 -28724.641} C_VEL
LIN {X 0,Y 56.07,Z 517.437,A -85,B 0,C 180,E1 -28734.991,E2 -28734.991} C_VEL
LIN {X 0,Y 55.631,Z 520.953,A -85,B 0,C 180,E1 -28744.625,E2 -28744.625} C_VEL
LIN {X 0,Y 57.382,Z 524.296,A -85,B 0,C 180,E1 -28757.271,E2 -28757.271} C_VEL
LIN {X 0,Y 59.939,Z 525.725,A -85,B 0,C 180,E1 -28765.134,E2 -28765.134} C_VEL
LIN {X 0,Y 64.719,Z 526.672,A -85,B 0,C 180,E1 -28774.257,E2 -28774.257} C_VEL
LIN {X 0,Y 71.676,Z 526.528,A -85,B 0,C 180,E1 -28782.895,E2 -28782.895} C_VEL
LIN {X 0,Y 79.791,Z 525.083,A -85,B 0,C 180,E1 -28789.856,E2 -28789.856} C_VEL
LIN {X 0,Y 88.97,Z 522.31,A -85,B 0,C 180,E1 -28795.471,E2 -28795.471} C_VEL
LIN {X 0,Y 98.985,Z 518.037,A -85,B 0,C 180,E1 -28800.001,E2 -28800.001} C_VEL
LIN {X 0,Y 102.039,Z 516.371,A -85,B 0,C 180,E1 -28801.975,E2 -28801.975} C_VEL
LIN {X 0,Y 102.858,Z 515.699,A -85,B 0,C 180,E1 -28803.919,E2 -28803.919} C_VEL
LIN {X 0,Y 104.099,Z 514.787,A -85,B 0,C 180,E1 -28807.761,E2 -28807.761} C_VEL
LIN {X 0,Y 104.215,Z 514.654,A -85,B 0,C 180,E1 -28811.674,E2 -28811.674} C_VEL
LIN {X 0,Y 104.111,Z 514.981,A -85,B 0,C 180,E1 -28815.667,E2 -28815.667} C_VEL
LIN {X 0,Y 103.604,Z 515.875,A -85,B 0,C 180,E1 -28819.828,E2 -28819.828} C_VEL
LIN {X 0,Y 102.902,Z 517.203,A -85,B 0,C 180,E1 -28824.193,E2 -28824.193} C_VEL
LIN {X 0,Y 102.169,Z 518.231,A -85,B 0,C 180,E1 -28826.611,E2 -28826.611} C_VEL
LIN {X 0,Y 99.526,Z 519.875,A -85,B 0,C 180,E1 -28828.054,E2 -28828.054} C_VEL
LIN {X 0,Y 90.721,Z 524.191,A -85,B 0,C 180,E1 -28831.574,E2 -28831.574} C_VEL
LIN {X 0,Y 85.164,Z 526.482,A -85,B 0,C 180,E1 -28834.409,E2 -28834.409} C_VEL
LIN {X 0,Y 77.693,Z 529.009,A -85,B 0,C 180,E1 -28839.29,E2 -28839.29} C_VEL
LIN {X 0,Y 70.449,Z 530.784,A -85,B 0,C 180,E1 -28845.727,E2 -28845.727} C_VEL
LIN {X 0,Y 66.351,Z 531.432,A -85,B 0,C 180,E1 -28850.56,E2 -28850.56} C_VEL
LIN {X 0,Y 59.902,Z 531.506,A -85,B 0,C 180,E1 -28862.029,E2 -28862.029} C_VEL
LIN {X 0,Y 57.821,Z 530.992,A -85,B 0,C 180,E1 -28868.632,E2 -28868.632} C_VEL
LIN {X 0,Y 56.546,Z 530.057,A -85,B 0,C 180,E1 -28875.623,E2 -28875.623} C_VEL
LIN {X 0,Y 56.738,Z 526.982,A -85,B 0,C 180,E1 -28890.016,E2 -28890.016} C_VEL
LIN {X 0,Y 57.137,Z 526.312,A -85,B 0,C 180,E1 -28892.88,E2 -28892.88} C_VEL
LIN {X 0,Y 57.52,Z 531.427,A -85,B 0,C 180,E1 -28904.16,E2 -28904.16} C_VEL
LIN {X 0,Y 60.734,Z 536.309,A -85,B 0,C 180,E1 -28917.588,E2 -28917.588} C_VEL
LIN {X 0,Y 66.978,Z 539.791,A -85,B 0,C 180,E1 -28929.035,E2 -28929.035} C_VEL
LIN {X 0,Y 75.752,Z 542.048,A -85,B 0,C 180,E1 -28937.936,E2 -28937.936} C_VEL
LIN {X 0,Y 86.106,Z 543.105,A -85,B 0,C 180,E1 -28944.722,E2 -28944.722} C_VEL
LIN {X 0,Y 97.489,Z 542.966,A -85,B 0,C 180,E1 -28949.908,E2 -28949.908} C_VEL
LIN {X 0,Y 98.938,Z 542.855,A -85,B 0,C 180,E1 -28950.448,E2 -28950.448} C_VEL
LIN {X 0,Y 100.486,Z 542.664,A -85,B 0,C 180,E1 -28952.009,E2 -28952.009} C_VEL
LIN {X 0,Y 89.098,Z 542.666,A -85,B 0,C 180,E1 -28956.77,E2 -28956.77} C_VEL
LIN {X 0,Y 81.875,Z 541.984,A -85,B 0,C 180,E1 -28960.803,E2 -28960.803} C_VEL
LIN {X 0,Y 71.636,Z 539.746,A -85,B 0,C 180,E1 -28968.892,E2 -28968.892} C_VEL
LIN {X 0,Y 63.061,Z 535.868,A -85,B 0,C 180,E1 -28979.998,E2 -28979.998} C_VEL
LIN {X 0,Y 58.728,Z 531.953,A -85,B 0,C 180,E1 -28989.909,E2 -28989.909} C_VEL
LIN {X 0,Y 56.177,Z 526.414,A -85,B 0,C 180,E1 -29002.041,E2 -29002.041} C_VEL
LIN {X 0,Y 55.992,Z 519.62,A -85,B 0,C 180,E1 -29014.388,E2 -29014.388} C_VEL
LIN {X 0,Y 57.091,Z 512.885,A -85,B 0,C 180,E1 -29024.089,E2 -29024.089} C_VEL
LIN {X 0,Y 59.306,Z 504.304,A -85,B 0,C 180,E1 -29033.646,E2 -29033.646} C_VEL
LIN {X 0,Y 62.666,Z 494.297,A -85,B 0,C 180,E1 -29042.024,E2 -29042.024} C_VEL
LIN {X 0,Y 66.825,Z 482.767,A -85,B 0,C 180,E1 -29049.002,E2 -29049.002} C_VEL
LIN {X 0,Y 67.273,Z 479.966,A -85,B 0,C 180,E1 -29050.574,E2 -29050.574} C_VEL
LIN {X 0,Y 68.089,Z 480.863,A -85,B 0,C 180,E1 -29051.948,E2 -29051.948} C_VEL
LIN {X 0,Y 72.608,Z 481.4,A -85,B 0,C 180,E1 -29055.444,E2 -29055.444} C_VEL
LIN {X 0,Y 73.845,Z 482.299,A -85,B 0,C 180,E1 -29056.856,E2 -29056.856} C_VEL
LIN {X 0,Y 72.833,Z 485.586,A -85,B 0,C 180,E1 -29058.86,E2 -29058.86} C_VEL
LIN {X 0,Y 68.299,Z 494.057,A -85,B 0,C 180,E1 -29064.081,E2 -29064.081} C_VEL
LIN {X 0,Y 63.282,Z 502.854,A -85,B 0,C 180,E1 -29071.83,E2 -29071.83} C_VEL
LIN {X 0,Y 61.128,Z 506.58,A -85,B 0,C 180,E1 -29076.12,E2 -29076.12} C_VEL
LIN {X 0,Y 58.719,Z 509.8,A -85,B 0,C 180,E1 -29080.264,E2 -29080.264} C_VEL
LIN {X 0,Y 53.635,Z 514.366,A -85,B 0,C 180,E1 -29087.617,E2 -29087.617} C_VEL
LIN {X 0,Y 49.409,Z 518.221,A -85,B 0,C 180,E1 -29096.741,E2 -29096.741} C_VEL
LIN {X 0,Y 48.514,Z 520.309,A -85,B 0,C 180,E1 -29103.182,E2 -29103.182} C_VEL
LIN {X 0,Y 49.634,Z 523.445,A -85,B 0,C 180,E1 -29115.044,E2 -29115.044} C_VEL
LIN {X 0,Y 53.611,Z 525.986,A -85,B 0,C 180,E1 -29128.377,E2 -29128.377} C_VEL
LIN {X 0,Y 59.993,Z 527.123,A -85,B 0,C 180,E1 -29139.535,E2 -29139.535} C_VEL
LIN {X 0,Y 67.692,Z 526.967,A -85,B 0,C 180,E1 -29148.018,E2 -29148.018} C_VEL
LIN {X 0,Y 77.553,Z 525.299,A -85,B 0,C 180,E1 -29155.282,E2 -29155.282} C_VEL
LIN {X 0,Y 86.525,Z 522.718,A -85,B 0,C 180,E1 -29160.002,E2 -29160.002} C_VEL
LIN {X 0,Y 93.805,Z 519.905,A -85,B 0,C 180,E1 -29162.966,E2 -29162.966} C_VEL
LIN {X 0,Y 96.27,Z 518.815,A -85,B 0,C 180,E1 -29164.188,E2 -29164.188} C_VEL
LIN {X 0,Y 97.756,Z 517.959,A -85,B 0,C 180,E1 -29168.268,E2 -29168.268} C_VEL
LIN {X 0,Y 97.847,Z 517.976,A -85,B 0,C 180,E1 -29172.445,E2 -29172.445} C_VEL
LIN {X 0,Y 97.632,Z 518.443,A -85,B 0,C 180,E1 -29176.736,E2 -29176.736} C_VEL
LIN {X 0,Y 96.856,Z 519.454,A -85,B 0,C 180,E1 -29181.274,E2 -29181.274} C_VEL
LIN {X 0,Y 95.884,Z 520.538,A -85,B 0,C 180,E1 -29184.448,E2 -29184.448} C_VEL
LIN {X 0,Y 87.215,Z 524.418,A -85,B 0,C 180,E1 -29187.6,E2 -29187.6} C_VEL
LIN {X 0,Y 81.362,Z 526.585,A -85,B 0,C 180,E1 -29190.279,E2 -29190.279} C_VEL
LIN {X 0,Y 70.481,Z 529.619,A -85,B 0,C 180,E1 -29197.111,E2 -29197.111} C_VEL
LIN {X 0,Y 65.539,Z 530.551,A -85,B 0,C 180,E1 -29201.377,E2 -29201.377} C_VEL
LIN {X 0,Y 56.996,Z 531.199,A -85,B 0,C 180,E1 -29211.958,E2 -29211.958} C_VEL
LIN {X 0,Y 53.704,Z 530.971,A -85,B 0,C 180,E1 -29218.456,E2 -29218.456} C_VEL
LIN {X 0,Y 49.71,Z 529.299,A -85,B 0,C 180,E1 -29233.594,E2 -29233.594} C_VEL
LIN {X 0,Y 49.318,Z 526.99,A -85,B 0,C 180,E1 -29246.014,E2 -29246.014} C_VEL
LIN {X 0,Y 50.335,Z 524.931,A -85,B 0,C 180,E1 -29254.481,E2 -29254.481} C_VEL
LIN {X 0,Y 50.878,Z 529.735,A -85,B 0,C 180,E1 -29266.056,E2 -29266.056} C_VEL
LIN {X 0,Y 54.656,Z 534.94,A -85,B 0,C 180,E1 -29280.972,E2 -29280.972} C_VEL
LIN {X 0,Y 61.687,Z 538.727,A -85,B 0,C 180,E1 -29293.143,E2 -29293.143} C_VEL
LIN {X 0,Y 71.217,Z 541.325,A -85,B 0,C 180,E1 -29302.155,E2 -29302.155} C_VEL
LIN {X 0,Y 82.216,Z 542.677,A -85,B 0,C 180,E1 -29308.759,E2 -29308.759} C_VEL
LIN {X 0,Y 88.055,Z 542.912,A -85,B 0,C 180,E1 -29311.415,E2 -29311.415} C_VEL
LIN {X 0,Y 87.748,Z 542.887,A -85,B 0,C 180,E1 -29311.785,E2 -29311.785} C_VEL
LIN {X 0,Y 75.964,Z 541.526,A -85,B 0,C 180,E1 -29317.722,E2 -29317.722} C_VEL
LIN {X 0,Y 65.159,Z 538.728,A -85,B 0,C 180,E1 -29326.155,E2 -29326.155} C_VEL
LIN {X 0,Y 56.276,Z 534.38,A -85,B 0,C 180,E1 -29337.9,E2 -29337.9} C_VEL
LIN {X 0,Y 51.254,Z 529.386,A -85,B 0,C 180,E1 -29350.492,E2 -29350.492} C_VEL
LIN {X 0,Y 49.129,Z 523.843,A -85,B 0,C 180,E1 -29363.163,E2 -29363.163} C_VEL
LIN {X 0,Y 49.291,Z 516.33,A -85,B 0,C 180,E1 -29377.295,E2 -29377.295} C_VEL
LIN {X 0,Y 51.021,Z 507.975,A -85,B 0,C 180,E1 -29389.372,E2 -29389.372} C_VEL
LIN {X 0,Y 54.255,Z 497.838,A -85,B 0,C 180,E1 -29400.179,E2 -29400.179} C_VEL
LIN {X 0,Y 58.26,Z 487.205,A -85,B 0,C 180,E1 -29408.257,E2 -29408.257} C_VEL
LIN {X 0,Y 58.785,Z 485.84,A -85,B 0,C 180,E1 -29409.138,E2 -29409.138} C_VEL
LIN {X 0,Y 59.596,Z 486.531,A -85,B 0,C 180,E1 -29410.626,E2 -29410.626} C_VEL
LIN {X 0,Y 65.463,Z 486.465,A -85,B 0,C 180,E1 -29415.059,E2 -29415.059} C_VEL
LIN {X 0,Y 66.207,Z 487.294,A -85,B 0,C 180,E1 -29416.323,E2 -29416.323} C_VEL
LIN {X 0,Y 61.508,Z 495.297,A -85,B 0,C 180,E1 -29421.772,E2 -29421.772} C_VEL
LIN {X 0,Y 56.222,Z 503.808,A -85,B 0,C 180,E1 -29430.124,E2 -29430.124} C_VEL
LIN {X 0,Y 51.783,Z 511.181,A -85,B 0,C 180,E1 -29440.945,E2 -29440.945} C_VEL
LIN {X 0,Y 49.502,Z 515.912,A -85,B 0,C 180,E1 -29450.769,E2 -29450.769} C_VEL
LIN {X 0,Y 48.514,Z 520.309,A -85,B 0,C 180,E1 -29463.182,E2 -29463.182} C_VEL
LIN {X 0,Y 48.191,Z 522.162,A -85,B 0,C 180,E1 -29469.812,E2 -29469.812} C_VEL
LIN {X 0,Y 47.337,Z 524.56,A -85,B 0,C 180,E1 -29481.317,E2 -29481.317} C_VEL
LIN {X 0,Y 47.948,Z 526.008,A -85,B 0,C 180,E1 -29490.72,E2 -29490.72} C_VEL
LIN {X 0,Y 49.955,Z 526.843,A -85,B 0,C 180,E1 -29497.178,E2 -29497.178} C_VEL
LIN {X 0,Y 50.987,Z 527.008,A -85,B 0,C 180,E1 -29499.07,E2 -29499.07} C_VEL
LIN {X 0,Y 57.553,Z 527.644,A -85,B 0,C 180,E1 -29507.583,E2 -29507.583} C_VEL
LIN {X 0,Y 64.323,Z 527.406,A -85,B 0,C 180,E1 -29513.729,E2 -29513.729} C_VEL
LIN {X 0,Y 74.123,Z 525.937,A -85,B 0,C 180,E1 -29520.002,E2 -29520.002} C_VEL
LIN {X 0,Y 84.699,Z 523.139,A -85,B 0,C 180,E1 -29524.761,E2 -29524.761} C_VEL
LIN {X 0,Y 90.213,Z 521.204,A -85,B 0,C 180,E1 -29526.712,E2 -29526.712} C_VEL
LIN {X 0,Y 91.246,Z 520.777,A -85,B 0,C 180,E1 -29528.863,E2 -29528.863} C_VEL
LIN {X 0,Y 91.243,Z 520.928,A -85,B 0,C 180,E1 -29533.362,E2 -29533.362} C_VEL
LIN {X 0,Y 90.814,Z 521.54,A -85,B 0,C 180,E1 -29538.034,E2 -29538.034} C_VEL
LIN {X 0,Y 90.228,Z 522.154,A -85,B 0,C 180,E1 -29540.852,E2 -29540.852} C_VEL
LIN {X 0,Y 87.309,Z 523.408,A -85,B 0,C 180,E1 -29542.257,E2 -29542.257} C_VEL
LIN {X 0,Y 78.019,Z 526.636,A -85,B 0,C 180,E1 -29545.766,E2 -29545.766} C_VEL
LIN {X 0,Y 67.966,Z 529.164,A -85,B 0,C 180,E1 -29551.135,E2 -29551.135} C_VEL
LIN {X 0,Y 61.067,Z 530.263,A -85,B 0,C 180,E1 -29556.358,E2 -29556.358} C_VEL
LIN {X 0,Y 51.584,Z 530.741,A -85,B 0,C 180,E1 -29567.086,E2 -29567.086} C_VEL
LIN {X 0,Y 44.87,Z 529.638,A -85,B 0,C 180,E1 -29581.996,E2 -29581.996} C_VEL
LIN {X 0,Y 42.942,Z 528.526,A -85,B 0,C 180,E1 -29590.916,E2 -29590.916} C_VEL
LIN {X 0,Y 42.286,Z 525.972,A -85,B 0,C 180,E1 -29605.771,E2 -29605.771} C_VEL
LIN {X 0,Y 43.543,Z 523.503,A -85,B 0,C 180,E1 -29616.682,E2 -29616.682} C_VEL
LIN {X 0,Y 45.075,Z 529.479,A -85,B 0,C 180,E1 -29632.963,E2 -29632.963} C_VEL
LIN {X 0,Y 50.557,Z 534.585,A -85,B 0,C 180,E1 -29648.744,E2 -29648.744} C_VEL
LIN {X 0,Y 56.786,Z 537.571,A -85,B 0,C 180,E1 -29657.973,E2 -29657.973} C_VEL
LIN {X 0,Y 67.128,Z 540.434,A -85,B 0,C 180,E1 -29666.906,E2 -29666.906} C_VEL
LIN {X 0,Y 72.823,Z 541.425,A -85,B 0,C 180,E1 -29670.315,E2 -29670.315} C_VEL
LIN {X 0,Y 74.492,Z 541.634,A -85,B 0,C 180,E1 -29671.852,E2 -29671.852} C_VEL
LIN {X 0,Y 61.877,Z 538.546,A -85,B 0,C 180,E1 -29680.076,E2 -29680.076} C_VEL
LIN {X 0,Y 53.738,Z 535.169,A -85,B 0,C 180,E1 -29688.684,E2 -29688.684} C_VEL
LIN {X 0,Y 47.388,Z 530.836,A -85,B 0,C 180,E1 -29699.997,E2 -29699.997} C_VEL
LIN {X 0,Y 42.998,Z 524.692,A -85,B 0,C 180,E1 -29715.728,E2 -29715.728} C_VEL
LIN {X 0,Y 42.026,Z 518.473,A -85,B 0,C 180,E1 -29730.108,E2 -29730.108} C_VEL
LIN {X 0,Y 42.663,Z 512.611,A -85,B 0,C 180,E1 -29741.214,E2 -29741.214} C_VEL
LIN {X 0,Y 44.779,Z 504.364,A -85,B 0,C 180,E1 -29753.544,E2 -29753.544} C_VEL
LIN {X 0,Y 48.286,Z 494.742,A -85,B 0,C 180,E1 -29764.09,E2 -29764.09} C_VEL
LIN {X 0,Y 49.573,Z 491.603,A -85,B 0,C 180,E1 -29767.027,E2 -29767.027} C_VEL
LIN {X 0,Y 52.028,Z 492.464,A -85,B 0,C 180,E1 -29771,E2 -29771} C_VEL
LIN {X 0,Y 57.355,Z 492.571,A -85,B 0,C 180,E1 -29775.798,E2 -29775.798} C_VEL
LIN {X 0,Y 51.404,Z 501.52,A -85,B 0,C 180,E1 -29783.994,E2 -29783.994} C_VEL
LIN {X 0,Y 46.404,Z 508.844,A -85,B 0,C 180,E1 -29794.324,E2 -29794.324} C_VEL
LIN {X 0,Y 43.026,Z 514.597,A -85,B 0,C 180,E1 -29806.326,E2 -29806.326} C_VEL
LIN {X 0,Y 41.421,Z 519.803,A -85,B 0,C 180,E1 -29821.972,E2 -29821.972} C_VEL
LIN {X 0,Y 43.21,Z 523.906,A -85,B 0,C 180,E1 -29839.418,E2 -29839.418} C_VEL
LIN {X 0,Y 48.221,Z 526.432,A -85,B 0,C 180,E1 -29854.076,E2 -29854.076} C_VEL
LIN {X 0,Y 50.987,Z 527.008,A -85,B 0,C 180,E1 -29859.07,E2 -29859.07} C_VEL
